KUKA KRL program: MyProgram_143().src

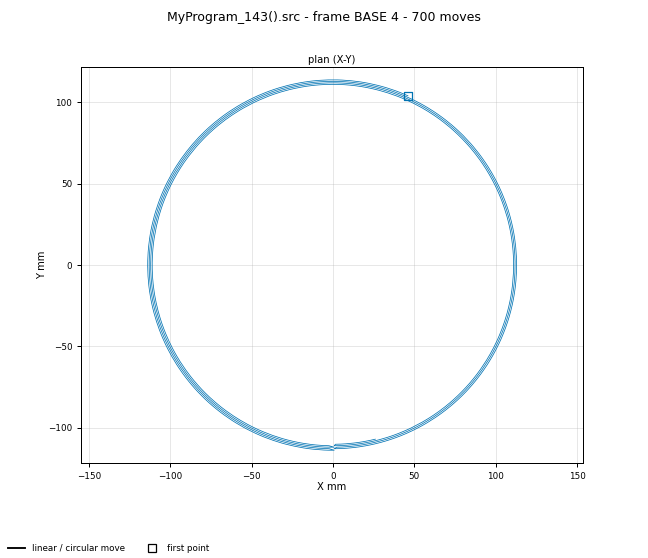
[picture p0: tool path of MyProgram_143().src in frame BASE 4, 700 of 700 moves have a stored position in this frame; points joined in program order, loops and branches not executed]
&ACCESS RVP
&REL 1
&PARAM TEMPLATE = C:\KRC\Roboter\Template\vorgabe
&PARAM EDITMASK = *
DEF MyProgram_143()
; ---- Setting reference (Base) ----
$BASE = BASE_DATA[4]

; --------------------------
; ---- Setting tool (TCP) ----
$TOOL = TOOL_DATA[3]
; --------------------------

$VEL.CP = VEL_APROX_PRINT
Startdeposition()
$VEL.CP = VEL_PRINT
LIN {X 46.1165,Y 104.0371,Z 114,A 62.0939,B 24.9325,C -1.8981,E1 25.0637,E2 383.7056} C_DIS
LIN {X 43.2178,Y 105.2725,Z 114,A 63.5467,B 24.9328,C -1.8939,E1 25.06,E2 382.2661} C_DIS
LIN {X 40.9561,Y 106.1746,Z 114,A 64.7702,B 24.9327,C -1.895,E1 25.0568,E2 381.0428} C_DIS
LIN {X 38.0003,Y 107.2663,Z 114,A 66.3534,B 24.9326,C -1.8963,E1 25.0527,E2 379.4597} C_DIS
LIN {X 35.3564,Y 108.1666,Z 114,A 67.7569,B 24.9326,C -1.8974,E1 25.0489,E2 378.0564} C_DIS
LIN {X 33.0344,Y 108.8999,Z 114,A 69.1112,B 24.932,C -1.9039,E1 25.0453,E2 376.689} C_DIS
LIN {X 30.3519,Y 109.6778,Z 114,A 70.5154,B 24.932,C -1.9048,E1 25.0415,E2 375.2851} C_DIS
LIN {X 27.6512,Y 110.3896,Z 114,A 71.9198,B 24.932,C -1.9055,E1 25.0377,E2 373.881} C_DIS
LIN {X 24.584,Y 111.1112,Z 114,A 73.211,B 24.9328,C -1.8936,E1 25.0343,E2 372.6199} C_DIS
LIN {X 22.2013,Y 111.6134,Z 114,A 74.5993,B 24.9322,C -1.9011,E1 25.0304,E2 371.2154} C_DIS
LIN {X 19.4555,Y 112.1246,Z 114,A 76.0045,B 24.9322,C -1.9016,E1 25.0266,E2 369.8105} C_DIS
LIN {X 16.6979,Y 112.5683,Z 114,A 77.5399,B 24.9318,C -1.9077,E1 25.0223,E2 368.2623} C_DIS
LIN {X 13.5748,Y 112.9859,Z 114,A 78.8318,B 24.9327,C -1.8953,E1 25.0188,E2 367.0007} C_DIS
LIN {X 11.1544,Y 113.2521,Z 114,A 80.3513,B 24.9317,C -1.9081,E1 25.0145,E2 365.4519} C_DIS
LIN {X 8.0145,Y 113.5158,Z 114,A 81.8072,B 24.9321,C -1.9026,E1 25.0105,E2 364.0098} C_DIS
LIN {X 5.5839,Y 113.663,Z 114,A 83.1636,B 24.9317,C -1.9081,E1 25.0067,E2 362.6407} C_DIS
LIN {X 2.7928,Y 113.7658,Z 114,A 84.4401,B 24.9322,C -1.9024,E1 25.0032,E2 361.3781} C_DIS
LIN {X -0.358,Y 113.7978,Z 114,A 86.0421,B 24.9322,C -1.9028,E1 24.9987,E2 359.7753} C_DIS
LIN {X -2.7928,Y 113.7658,Z 114,A 87.3841,B 24.9318,C -1.9074,E1 24.9949,E2 358.4222} C_DIS
LIN {X -5.7875,Y 113.6517,Z 114,A 88.6706,B 24.9325,C -1.8975,E1 24.9914,E2 357.159} C_DIS
LIN {X -8.3717,Y 113.4917,Z 114,A 90.1989,B 24.9319,C -1.9064,E1 24.9871,E2 355.6088} C_DIS
LIN {X -11.5104,Y 113.2148,Z 114,A 91.4931,B 24.9328,C -1.8933,E1 24.9835,E2 354.3452} C_DIS
LIN {X -14.2853,Y 112.8982,Z 114,A 93.065,B 24.9324,C -1.8995,E1 24.9791,E2 352.7575} C_DIS
LIN {X -17.0517,Y 112.5136,Z 114,A 94.473,B 24.9324,C -1.8986,E1 24.9753,E2 351.3504} C_DIS
LIN {X -19.8078,Y 112.0613,Z 114,A 95.8815,B 24.9324,C -1.8977,E1 24.9714,E2 349.9428} C_DIS
LIN {X -22.5519,Y 111.5414,Z 114,A 97.3152,B 24.9324,C -1.8977,E1 24.9674,E2 348.5075} C_DIS
LIN {X -24.9337,Y 111.0349,Z 114,A 98.5186,B 24.9326,C -1.8956,E1 24.9642,E2 347.3074} C_DIS
LIN {X -28.04,Y 110.2897,Z 114,A 100.1157,B 24.9328,C -1.8936,E1 24.9598,E2 345.7129} C_DIS
LIN {X -30.7893,Y 109.5538,Z 114,A 101.5344,B 24.9329,C -1.8915,E1 24.956,E2 344.2969} C_DIS
LIN {X -33.3763,Y 108.7938,Z 114,A 102.9287,B 24.9329,C -1.8915,E1 24.9523,E2 342.9003} C_DIS
LIN {X -36.0362,Y 107.942,Z 114,A 104.1731,B 24.9335,C -1.8831,E1 24.949,E2 341.6736} C_DIS
LIN {X -38.6744,Y 107.0251,Z 114,A 105.7474,B 24.9332,C -1.8883,E1 24.9449,E2 340.0839} C_DIS
LIN {X -41.2893,Y 106.0437,Z 114,A 107.1576,B 24.9332,C -1.8866,E1 24.9412,E2 338.6748} C_DIS
LIN {X -43.8793,Y 104.9985,Z 114,A 108.5683,B 24.9334,C -1.8848,E1 24.9375,E2 337.2652} C_DIS
LIN {X -46.1165,Y 104.0371,Z 114,A 109.7983,B 24.9335,C -1.8831,E1 24.9344,E2 336.0362} C_DIS
LIN {X -48.6835,Y 102.8607,Z 114,A 111.3437,B 24.9333,C -1.886,E1 24.9305,E2 334.4801} C_DIS
LIN {X -51.4845,Y 101.4861,Z 114,A 112.8012,B 24.9338,C -1.8788,E1 24.9269,E2 333.0359} C_DIS
LIN {X -53.9596,Y 100.192,Z 114,A 114.2127,B 24.934,C -1.8767,E1 24.9234,E2 331.6255} C_DIS
LIN {X -56.0918,Y 99.0159,Z 114,A 115.4434,B 24.9341,C -1.8747,E1 24.9204,E2 330.3961} C_DIS
LIN {X -58.8108,Y 97.4236,Z 114,A 117.036,B 24.9343,C -1.8721,E1 24.9166,E2 328.8048} C_DIS
LIN {X -61.184,Y 95.951,Z 114,A 118.2834,B 24.9349,C -1.8629,E1 24.9137,E2 327.5752} C_DIS
LIN {X -63.2239,Y 94.6213,Z 114,A 119.8102,B 24.9343,C -1.8728,E1 24.91,E2 326.0199} C_DIS
LIN {X -65.8184,Y 92.8333,Z 114,A 121.2145,B 24.935,C -1.8622,E1 24.9069,E2 324.636} C_DIS
LIN {X -68.0768,Y 91.1901,Z 114,A 122.5208,B 24.9355,C -1.8552,E1 24.904,E2 323.3418} C_DIS
LIN {X -70.2942,Y 89.4919,Z 114,A 124.098,B 24.9352,C -1.8591,E1 24.9004,E2 321.7495} C_DIS
LIN {X -72.194,Y 87.9686,Z 114,A 125.3301,B 24.9354,C -1.8566,E1 24.8978,E2 320.5187} C_DIS
LIN {X -74.3311,Y 86.1704,Z 114,A 126.874,B 24.9352,C -1.859,E1 24.8945,E2 318.963} C_DIS
LIN {X -76.4234,Y 84.3203,Z 114,A 128.1561,B 24.9358,C -1.8507,E1 24.8918,E2 317.6955} C_DIS
LIN {X -78.4697,Y 82.4194,Z 114,A 129.7007,B 24.9356,C -1.853,E1 24.8887,E2 316.1392} C_DIS
LIN {X -80.7204,Y 80.2141,Z 114,A 131.1644,B 24.9362,C -1.8442,E1 24.8858,E2 314.6902} C_DIS
LIN {X -82.4194,Y 78.4697,Z 114,A 132.564,B 24.936,C -1.8482,E1 24.8831,E2 313.2751} C_DIS
LIN {X -84.559,Y 76.1567,Z 114,A 133.9922,B 24.9367,C -1.8378,E1 24.8804,E2 311.8653} C_DIS
LIN {X -86.1704,Y 74.3311,Z 114,A 135.2253,B 24.9369,C -1.8349,E1 24.8782,E2 310.6336} C_DIS
LIN {X -88.194,Y 71.9159,Z 114,A 136.6561,B 24.9376,C -1.8245,E1 24.8756,E2 309.2209} C_DIS
LIN {X -89.7139,Y 70.0134,Z 114,A 138.0538,B 24.9374,C -1.8281,E1 24.8732,E2 307.8081} C_DIS
LIN {X -91.6165,Y 67.5018,Z 114,A 139.4849,B 24.9381,C -1.8176,E1 24.8708,E2 306.3952} C_DIS
LIN {X -93.0412,Y 65.527,Z 114,A 141.0139,B 24.9375,C -1.8263,E1 24.8683,E2 304.8379} C_DIS
LIN {X -94.8183,Y 62.9251,Z 114,A 142.4789,B 24.9381,C -1.817,E1 24.866,E2 303.3877} C_DIS
LIN {X -96.1444,Y 60.8828,Z 114,A 143.8436,B 24.938,C -1.8191,E1 24.864,E2 302.0113} C_DIS
LIN {X -97.6096,Y 58.5049,Z 114,A 145.1278,B 24.9386,C -1.8101,E1 24.8621,E2 300.7418} C_DIS
LIN {X -99.1905,Y 55.7793,Z 114,A 146.5592,B 24.9393,C -1.7993,E1 24.8602,E2 299.3286} C_DIS
LIN {X -100.5295,Y 53.3282,Z 114,A 147.9748,B 24.9396,C -1.7956,E1 24.8583,E2 297.9145} C_DIS
LIN {X -101.649,Y 51.1658,Z 114,A 149.3733,B 24.9394,C -1.7988,E1 24.8565,E2 296.501} C_DIS
LIN {X -102.874,Y 48.6558,Z 114,A 150.7887,B 24.9396,C -1.7949,E1 24.8548,E2 295.0871} C_DIS
LIN {X -104.0371,Y 46.1165,Z 114,A 152.3355,B 24.9396,C -1.7962,E1 24.853,E2 293.5286} C_DIS
LIN {X -105.1375,Y 43.5494,Z 114,A 153.6201,B 24.9401,C -1.787,E1 24.8516,E2 292.2588} C_DIS
LIN {X -106.1746,Y 40.9561,Z 114,A 155.0356,B 24.9404,C -1.7831,E1 24.8502,E2 290.8448} C_DIS
LIN {X -107.2085,Y 38.1651,Z 114,A 156.6062,B 24.9405,C -1.7813,E1 24.8487,E2 289.2696} C_DIS
LIN {X -108.1666,Y 35.3564,Z 114,A 157.8837,B 24.9414,C -1.768,E1 24.8476,E2 288.0165} C_DIS
LIN {X -108.8999,Y 33.0344,Z 114,A 159.2832,B 24.9412,C -1.771,E1 24.8464,E2 286.6019} C_DIS
LIN {X -109.7859,Y 29.9514,Z 114,A 160.7183,B 24.942,C -1.7587,E1 24.8453,E2 285.1876} C_DIS
LIN {X -110.4745,Y 27.3034,Z 114,A 162.1316,B 24.9422,C -1.7557,E1 24.8444,E2 283.7732} C_DIS
LIN {X -111.1112,Y 24.584,Z 114,A 163.7041,B 24.9421,C -1.7578,E1 24.8434,E2 282.1865} C_DIS
LIN {X -111.6811,Y 21.8498,Z 114,A 165.1331,B 24.9423,C -1.7542,E1 24.8426,E2 280.7577} C_DIS
LIN {X -112.1837,Y 19.1024,Z 114,A 166.3797,B 24.943,C -1.7433,E1 24.842,E2 279.5296} C_DIS
LIN {X -112.6187,Y 16.3435,Z 114,A 167.7956,B 24.9433,C -1.7391,E1 24.8414,E2 278.1152} C_DIS
LIN {X -112.9859,Y 13.5748,Z 114,A 169.2121,B 24.9436,C -1.735,E1 24.8409,E2 276.7003} C_DIS
LIN {X -113.2521,Y 11.1544,Z 114,A 170.6117,B 24.9434,C -1.7379,E1 24.8405,E2 275.2854} C_DIS
LIN {X -113.5158,Y 8.0145,Z 114,A 172.209,B 24.9437,C -1.7332,E1 24.8401,E2 273.6896} C_DIS
LIN {X -113.6762,Y 5.2757,Z 114,A 173.6173,B 24.9439,C -1.7297,E1 24.8399,E2 272.2811} C_DIS
LIN {X -113.7658,Y 2.7928,Z 114,A 175.0421,B 24.9437,C -1.7326,E1 24.8399,E2 270.8409} C_DIS
LIN {X -113.7945,Y -0.969,Z 114,A 176.8249,B 24.9444,C -1.722,E1 24.8399,E2 269.0726} C_DIS
LIN {X -113.7006,Y -4.7094,Z 114,A 178.4247,B 24.9455,C -1.7046,E1 24.8399,E2 267.5046} C_DIS
LIN {X -113.5859,Y -6.9783,Z 114,A 179.9475,B 24.9448,C -1.716,E1 24.8402,E2 265.9456} C_DIS
LIN {X -113.3475,Y -10.1202,Z 114,A -178.5862,B 24.9455,C -1.7061,E1 24.8405,E2 264.494} C_DIS
LIN {X -113.1067,Y -12.5433,Z 114,A -177.2205,B 24.9453,C -1.7077,E1 24.8409,E2 263.1162} C_DIS
LIN {X -112.7144,Y -15.6697,Z 114,A -175.7543,B 24.946,C -1.6979,E1 24.8415,E2 261.6647} C_DIS
LIN {X -112.2959,Y -18.4311,Z 114,A -174.503,B 24.9466,C -1.6873,E1 24.842,E2 260.4313} C_DIS
LIN {X -111.8774,Y -20.8299,Z 114,A -172.9727,B 24.9461,C -1.6955,E1 24.8428,E2 258.8723} C_DIS
LIN {X -111.3326,Y -23.5693,Z 114,A -171.5211,B 24.9463,C -1.6929,E1 24.8436,E2 257.4183} C_DIS
LIN {X -110.7206,Y -26.2944,Z 114,A -170.1412,B 24.9466,C -1.6875,E1 24.8445,E2 256.0432} C_DIS
LIN {X -109.9486,Y -29.3493,Z 114,A -168.6752,B 24.9472,C -1.6778,E1 24.8455,E2 254.5919} C_DIS
LIN {X -109.1952,Y -32.0387,Z 114,A -167.4243,B 24.9479,C -1.6673,E1 24.8464,E2 253.3588} C_DIS
LIN {X -108.3987,Y -34.639,Z 114,A -166.0121,B 24.9481,C -1.6648,E1 24.8476,E2 251.9442} C_DIS
LIN {X -107.6102,Y -37.0203,Z 114,A -164.61,B 24.948,C -1.6666,E1 24.8489,E2 250.53} C_DIS
LIN {X -106.6692,Y -39.6501,Z 114,A -163.0638,B 24.9479,C -1.668,E1 24.8504,E2 248.9716} C_DIS
LIN {X -105.5291,Y -42.5875,Z 114,A -161.5985,B 24.9485,C -1.6585,E1 24.8519,E2 247.5207} C_DIS
LIN {X -104.4521,Y -45.1645,Z 114,A -160.1215,B 24.9485,C -1.6573,E1 24.8535,E2 246.0385} C_DIS
LIN {X -102.874,Y -48.6558,Z 114,A -158.1112,B 24.9487,C -1.655,E1 24.8559,E2 244.0226} C_DIS
LIN {X -101.4861,Y -51.4845,Z 114,A -156.6461,B 24.9492,C -1.6457,E1 24.8577,E2 242.5718} C_DIS
LIN {X -100.192,Y -53.9596,Z 114,A -155.2312,B 24.9495,C -1.6422,E1 24.8595,E2 241.1579} C_DIS
LIN {X -99.0159,Y -56.0918,Z 114,A -153.998,B 24.9497,C -1.6391,E1 24.8612,E2 239.9256} C_DIS
LIN {X -97.3228,Y -58.9767,Z 114,A -152.3668,B 24.9501,C -1.6325,E1 24.8635,E2 238.3017} C_DIS
LIN {X -95.951,Y -61.184,Z 114,A -151.1167,B 24.9504,C -1.6267,E1 24.8654,E2 237.0591} C_DIS
LIN {X -94.6213,Y -63.2239,Z 114,A -149.6243,B 24.95,C -1.6343,E1 24.8677,E2 235.541} C_DIS
LIN {X -92.2301,Y -66.6638,Z 114,A -147.5035,B 24.9502,C -1.6295,E1 24.8711,E2 233.4214} C_DIS
LIN {X -90.5663,Y -68.9072,Z 114,A -146.09,B 24.9504,C -1.6263,E1 24.8735,E2 232.0086} C_DIS
LIN {X -88.8479,Y -71.109,Z 114,A -144.8071,B 24.951,C -1.6179,E1 24.8757,E2 230.7398} C_DIS
LIN {X -86.8439,Y -73.5405,Z 114,A -143.377,B 24.9516,C -1.6078,E1 24.8782,E2 229.3271} C_DIS
LIN {X -85.013,Y -75.6497,Z 114,A -141.7994,B 24.9513,C -1.6116,E1 24.8812,E2 227.7334} C_DIS
LIN {X -83.1309,Y -77.7132,Z 114,A -140.3002,B 24.9513,C -1.6122,E1 24.884,E2 226.2259} C_DIS
LIN {X -80.4688,Y -80.4688,Z 114,A -138.4479,B 24.9517,C -1.6049,E1 24.8876,E2 224.3833} C_DIS
LIN {X -78.4697,Y -82.4194,Z 114,A -137.0355,B 24.9519,C -1.6022,E1 24.8905,E2 222.9714} C_DIS
LIN {X -76.4234,Y -84.3203,Z 114,A -135.4925,B 24.9517,C -1.605,E1 24.8937,E2 221.4155} C_DIS
LIN {X -74.3311,Y -86.1704,Z 114,A -134.0244,B 24.9517,C -1.6048,E1 24.8968,E2 219.9421} C_DIS
LIN {X -71.109,Y -88.8479,Z 114,A -131.9623,B 24.9521,C -1.5989,E1 24.9012,E2 217.8863} C_DIS
LIN {X -68.9072,Y -90.5663,Z 114,A -130.5508,B 24.9522,C -1.5966,E1 24.9044,E2 216.4751} C_DIS
LIN {X -66.6638,Y -92.2301,Z 114,A -129.2697,B 24.9527,C -1.5889,E1 24.9072,E2 215.2078} C_DIS
LIN {X -64.0839,Y -94.039,Z 114,A -127.6777,B 24.9528,C -1.5865,E1 24.9109,E2 213.6161} C_DIS
LIN {X -62.058,Y -95.39,Z 114,A -126.4471,B 24.9529,C -1.5848,E1 24.9137,E2 212.3856} C_DIS
LIN {X -59.6983,Y -96.8843,Z 114,A -124.906,B 24.9527,C -1.5883,E1 24.9174,E2 210.8313} C_DIS
LIN {X -56.9923,Y -98.4985,Z 114,A -123.6091,B 24.9536,C -1.5739,E1 24.9205,E2 209.5648} C_DIS
LIN {X -54.8725,Y -99.6968,Z 114,A -122.2152,B 24.9533,C -1.5792,E1 24.9239,E2 208.1543} C_DIS
LIN {X -52.4093,Y -101.0134,Z 114,A -120.8052,B 24.9533,C -1.5775,E1 24.9274,E2 206.7443} C_DIS
LIN {X -49.5919,Y -102.4242,Z 114,A -119.3037,B 24.9537,C -1.572,E1 24.9311,E2 205.2519} C_DIS
LIN {X -47.3897,Y -103.4634,Z 114,A -117.9855,B 24.9536,C -1.5744,E1 24.9345,E2 203.9246} C_DIS
LIN {X -44.8363,Y -104.5952,Z 114,A -116.5759,B 24.9536,C -1.573,E1 24.9381,E2 202.515} C_DIS
LIN {X -42.2559,Y -105.664,Z 114,A -115.0363,B 24.9534,C -1.5773,E1 24.9421,E2 200.9619} C_DIS
LIN {X -39.0676,Y -106.8817,Z 114,A -113.4085,B 24.9537,C -1.5719,E1 24.9464,E2 199.3436} C_DIS
LIN {X -36.6811,Y -107.7245,Z 114,A -112.1681,B 24.9539,C -1.5694,E1 24.9496,E2 198.1068} C_DIS
LIN {X -34.0264,Y -108.5923,Z 114,A -110.9232,B 24.9543,C -1.5614,E1 24.9529,E2 196.8785} C_DIS
LIN {X -31.6956,Y -109.297,Z 114,A -109.4288,B 24.9537,C -1.572,E1 24.957,E2 195.3565} C_DIS
LIN {X -29.0037,Y -110.042,Z 114,A -107.9933,B 24.9537,C -1.5724,E1 24.9609,E2 193.9179} C_DIS
LIN {X -25.9456,Y -110.8012,Z 114,A -106.5353,B 24.9541,C -1.566,E1 24.9648,E2 192.473} C_DIS
LIN {X -23.5693,Y -111.3326,Z 114,A -105.1778,B 24.9538,C -1.5711,E1 24.9685,E2 191.1018} C_DIS
LIN {X -20.4423,Y -111.9472,Z 114,A -103.8822,B 24.9546,C -1.5572,E1 24.972,E2 189.8378} C_DIS
LIN {X -18.0781,Y -112.3549,Z 114,A -102.4935,B 24.9541,C -1.5646,E1 24.9759,E2 188.4303} C_DIS
LIN {X -15.3153,Y -112.7648,Z 114,A -100.9564,B 24.9538,C -1.57,E1 24.9801,E2 186.8792} C_DIS
LIN {X -11.9787,Y -113.1658,Z 114,A -99.452,B 24.9543,C -1.5616,E1 24.9843,E2 185.3937} C_DIS
LIN {X -8.0145,Y -113.5158,Z 114,A -97.3901,B 24.9542,C -1.5641,E1 24.99,E2 183.325} C_DIS
LIN {X -5.5839,Y -113.663,Z 114,A -96.0341,B 24.9538,C -1.5698,E1 24.9939,E2 181.955} C_DIS
LIN {X -2.7928,Y -113.7658,Z 114,A -94.7582,B 24.9542,C -1.5643,E1 24.9974,E2 180.692} C_DIS
LIN {X 0.7991,Y -113.7938,Z 114,A -93.1524,B 24.9546,C -1.5559,E1 25.0018,E2 179.1062} C_DIS
Enddeposition()
LIN {X 0.7991,Y -113.7938,Z 114,A -93.1524,B 24.9546,C -1.5559,E1 25.0018,E2 179.1062} C_DIS
Startdeposition()
$VEL.CP = VEL_PRINT
LIN {X -2.2586,Y -112.8565,Z 114,A -95.1963,B 24.955,C -1.5503,E1 24.9961,E2 181.1633} C_DIS
LIN {X -9.0135,Y -112.5185,Z 114,A -98.6101,B 24.955,C -1.551,E1 24.9866,E2 184.5765} C_DIS
LIN {X -13.6469,Y -112.0522,Z 114,A -100.9708,B 24.955,C -1.5513,E1 24.98,E2 186.9379} C_DIS
LIN {X -18.5418,Y -111.3457,Z 114,A -103.5657,B 24.955,C -1.5484,E1 24.9728,E2 189.5418} C_DIS
LIN {X -22.4378,Y -110.6268,Z 114,A -105.6155,B 24.9551,C -1.5475,E1 24.9672,E2 191.596} C_DIS
LIN {X -26.0122,Y -109.8427,Z 114,A -107.4525,B 24.9551,C -1.5493,E1 24.9622,E2 193.4312} C_DIS
LIN {X -29.3354,Y -109.0005,Z 114,A -109.1292,B 24.9548,C -1.553,E1 24.9577,E2 195.1015} C_DIS
LIN {X -31.7632,Y -108.3185,Z 114,A -110.5257,B 24.955,C -1.549,E1 24.9539,E2 196.5098} C_DIS
LIN {X -35.5601,Y -107.1328,Z 114,A -112.4447,B 24.9547,C -1.5547,E1 24.9488,E2 198.4187} C_DIS
LIN {X -38.7299,Y -106.0267,Z 114,A -114.1848,B 24.9547,C -1.5547,E1 24.9442,E2 200.1622} C_DIS
LIN {X -42.313,Y -104.6487,Z 114,A -116.1255,B 24.9546,C -1.557,E1 24.9392,E2 202.1019} C_DIS
LIN {X -46.2152,Y -102.9847,Z 114,A -118.2734,B 24.9544,C -1.5595,E1 24.9337,E2 204.2487} C_DIS
LIN {X -48.99,Y -101.694,Z 114,A -119.7945,B 24.9542,C -1.5627,E1 24.9298,E2 205.7662} C_DIS
LIN {X -52.1714,Y -100.1002,Z 114,A -121.6226,B 24.9542,C -1.5641,E1 24.9253,E2 207.5959} C_DIS
LIN {X -54.6205,Y -98.7851,Z 114,A -123.1671,B 24.9544,C -1.5605,E1 24.9215,E2 209.1532} C_DIS
LIN {X -58.226,Y -96.7038,Z 114,A -125.2381,B 24.9541,C -1.5653,E1 24.9165,E2 211.2192} C_DIS
LIN {X -61.5631,Y -94.6156,Z 114,A -127.1227,B 24.9536,C -1.573,E1 24.9121,E2 213.0914} C_DIS
LIN {X -63.5831,Y -93.2683,Z 114,A -128.4203,B 24.9536,C -1.5724,E1 24.9091,E2 214.3948} C_DIS
LIN {X -66.6222,Y -91.1216,Z 114,A -130.2576,B 24.9534,C -1.5777,E1 24.9049,E2 216.2259} C_DIS
LIN {X -69.0307,Y -89.311,Z 114,A -131.7931,B 24.9532,C -1.5802,E1 24.9015,E2 217.761} C_DIS
LIN {X -71.4837,Y -87.3615,Z 114,A -133.5417,B 24.9534,C -1.5767,E1 24.8977,E2 219.5244} C_DIS
LIN {X -74.0275,Y -85.2155,Z 114,A -135.1616,B 24.9531,C -1.5828,E1 24.8943,E2 221.1361} C_DIS
LIN {X -76.6052,Y -82.9063,Z 114,A -136.8906,B 24.9528,C -1.5875,E1 24.8907,E2 222.861} C_DIS
LIN {X -79.2467,Y -80.3843,Z 114,A -138.7926,B 24.9527,C -1.5894,E1 24.8869,E2 224.7663} C_DIS
LIN {X -81.9311,Y -77.6476,Z 114,A -140.7693,B 24.9525,C -1.5924,E1 24.883,E2 226.7444} C_DIS
LIN {X -84.589,Y -74.7448,Z 114,A -142.8598,B 24.9525,C -1.5932,E1 24.8791,E2 228.8423} C_DIS
LIN {X -87.2958,Y -71.5648,Z 114,A -145.0018,B 24.9522,C -1.5973,E1 24.8753,E2 230.9844} C_DIS
LIN {X -89.4995,Y -68.786,Z 114,A -146.6681,B 24.9516,C -1.607,E1 24.8724,E2 232.6355} C_DIS
LIN {X -91.6911,Y -65.8371,Z 114,A -148.3274,B 24.9508,C -1.6198,E1 24.8697,E2 234.2722} C_DIS
LIN {X -93.0166,Y -63.9524,Z 114,A -149.7858,B 24.9514,C -1.6113,E1 24.8674,E2 235.7581} C_DIS
LIN {X -94.5965,Y -61.5921,Z 114,A -151.1105,B 24.9508,C -1.6196,E1 24.8654,E2 237.0696} C_DIS
LIN {X -96.2719,Y -58.9366,Z 114,A -152.8227,B 24.9508,C -1.6192,E1 24.8628,E2 238.7916} C_DIS
LIN {X -98.1671,Y -55.7247,Z 114,A -154.6317,B 24.9504,C -1.6276,E1 24.8603,E2 240.59} C_DIS
LIN {X -100.8755,Y -50.6571,Z 114,A -157.6127,B 24.95,C -1.6331,E1 24.8564,E2 243.5737} C_DIS
LIN {X -102.3686,Y -47.564,Z 114,A -159.3935,B 24.9498,C -1.6366,E1 24.8543,E2 245.3558} C_DIS
LIN {X -103.7319,Y -44.5169,Z 114,A -161.1653,B 24.9497,C -1.6384,E1 24.8523,E2 247.1331} C_DIS
LIN {X -104.9067,Y -41.6706,Z 114,A -162.6469,B 24.9492,C -1.6462,E1 24.8507,E2 248.6044} C_DIS
LIN {X -105.9693,Y -38.8872,Z 114,A -164.1989,B 24.949,C -1.6491,E1 24.8492,E2 250.1582} C_DIS
LIN {X -107.043,Y -35.8264,Z 114,A -165.8973,B 24.9489,C -1.652,E1 24.8477,E2 251.8594} C_DIS
LIN {X -108.0614,Y -32.6277,Z 114,A -168.1598,B 24.9499,C -1.6355,E1 24.8458,E2 254.1742} C_DIS
LIN {X -109.2232,Y -28.4979,Z 114,A -169.7983,B 24.9482,C -1.6631,E1 24.8447,E2 255.7565} C_DIS
LIN {X -110.1558,Y -24.6524,Z 114,A -171.7438,B 24.9476,C -1.6718,E1 24.8434,E2 257.6927} C_DIS
LIN {X -110.7486,Y -21.8326,Z 114,A -173.0922,B 24.9471,C -1.6808,E1 24.8427,E2 259.0275} C_DIS
LIN {X -111.2957,Y -18.841,Z 114,A -174.626,B 24.9467,C -1.6861,E1 24.8419,E2 260.5579} C_DIS
LIN {X -111.7711,Y -15.7763,Z 114,A -176.4489,B 24.947,C -1.6814,E1 24.8412,E2 262.4027} C_DIS
LIN {X -112.2153,Y -12.2317,Z 114,A -178.0389,B 24.9461,C -1.6959,E1 24.8407,E2 263.9678} C_DIS
LIN {X -112.5139,Y -9.0719,Z 114,A -179.8355,B 24.9462,C -1.6939,E1 24.8402,E2 265.78} C_DIS
LIN {X -112.7457,Y -5.5256,Z 114,A 178.2019,B 24.9462,C -1.6935,E1 24.8399,E2 267.7553} C_DIS
LIN {X -112.8722,Y -1.397,Z 114,A 176.1161,B 24.9458,C -1.7007,E1 24.8398,E2 269.8364} C_DIS
LIN {X -112.8551,Y 2.3368,Z 114,A 174.3952,B 24.945,C -1.7136,E1 24.8398,E2 271.5369} C_DIS
LIN {X -112.7327,Y 5.7632,Z 114,A 172.7548,B 24.9444,C -1.7231,E1 24.84,E2 273.1644} C_DIS
LIN {X -112.5317,Y 8.8494,Z 114,A 170.9857,B 24.9445,C -1.7205,E1 24.8404,E2 274.9504} C_DIS
LIN {X -112.1713,Y 12.6301,Z 114,A 169.0198,B 24.9442,C -1.7253,E1 24.8409,E2 276.9168} C_DIS
LIN {X -111.6851,Y 16.382,Z 114,A 167.0194,B 24.944,C -1.7284,E1 24.8417,E2 278.9217} C_DIS
LIN {X -111.1787,Y 19.5236,Z 114,A 165.3457,B 24.9438,C -1.7314,E1 24.8425,E2 280.5982} C_DIS
LIN {X -110.3652,Y 23.6924,Z 114,A 163.2697,B 24.9432,C -1.7414,E1 24.8437,E2 282.6625} C_DIS
LIN {X -109.5151,Y 27.3588,Z 114,A 161.1089,B 24.9434,C -1.7379,E1 24.8451,E2 284.8445} C_DIS
LIN {X -108.2752,Y 31.9089,Z 114,A 159.1024,B 24.9419,C -1.7605,E1 24.8466,E2 286.8087} C_DIS
LIN {X -107.2912,Y 35.0758,Z 114,A 157.205,B 24.9421,C -1.7575,E1 24.8482,E2 288.7242} C_DIS
LIN {X -106.422,Y 37.6311,Z 114,A 155.3289,B 24.9431,C -1.7422,E1 24.85,E2 290.6472} C_DIS
LIN {X -104.9357,Y 41.5967,Z 114,A 153.3141,B 24.9423,C -1.7541,E1 24.8521,E2 292.6452} C_DIS
LIN {X -103.5701,Y 44.8882,Z 114,A 151.811,B 24.9412,C -1.7714,E1 24.8537,E2 294.1152} C_DIS
LIN {X -101.9941,Y 48.3653,Z 114,A 150.106,B 24.9402,C -1.7863,E1 24.8556,E2 295.7941} C_DIS
LIN {X -100.589,Y 51.2206,Z 114,A 148.4035,B 24.9401,C -1.7877,E1 24.8578,E2 297.5022} C_DIS
LIN {X -99.0805,Y 54.0815,Z 114,A 146.6333,B 24.9401,C -1.7876,E1 24.8601,E2 299.2822} C_DIS
LIN {X -97.4137,Y 57.0303,Z 114,A 144.5089,B 24.9408,C -1.7769,E1 24.8632,E2 301.4431} C_DIS
LIN {X -95.5003,Y 60.1794,Z 114,A 143.0585,B 24.9394,C -1.7985,E1 24.8652,E2 302.8494} C_DIS
LIN {X -93.6718,Y 62.9873,Z 114,A 141.3181,B 24.9392,C -1.8017,E1 24.8679,E2 304.5908} C_DIS
LIN {X -91.4817,Y 66.1305,Z 114,A 139.328,B 24.9389,C -1.8053,E1 24.8711,E2 306.5821} C_DIS
LIN {X -89.4267,Y 68.8806,Z 114,A 137.7955,B 24.938,C -1.8183,E1 24.8737,E2 308.091} C_DIS
LIN {X -87.085,Y 71.8196,Z 114,A 135.6803,B 24.9382,C -1.8152,E1 24.8774,E2 310.2235} C_DIS
LIN {X -84.6596,Y 74.664,Z 114,A 133.7205,B 24.9381,C -1.8176,E1 24.881,E2 312.1863} C_DIS
LIN {X -81.997,Y 77.5775,Z 114,A 131.7125,B 24.9377,C -1.8225,E1 24.8848,E2 314.1915} C_DIS
LIN {X -79.2984,Y 80.3332,Z 114,A 129.8833,B 24.9371,C -1.8323,E1 24.8884,E2 316.0051} C_DIS
LIN {X -76.5557,Y 82.9518,Z 114,A 127.8785,B 24.937,C -1.8337,E1 24.8925,E2 318.0148} C_DIS
LIN {X -73.5611,Y 85.6192,Z 114,A 125.8041,B 24.9368,C -1.8368,E1 24.8968,E2 320.09} C_DIS
LIN {X -71.2356,Y 87.5626,Z 114,A 124.4734,B 24.936,C -1.8485,E1 24.8997,E2 321.398} C_DIS
LIN {X -68.5761,Y 89.6613,Z 114,A 122.5677,B 24.9362,C -1.8447,E1 24.9039,E2 323.3196} C_DIS
LIN {X -65.7243,Y 91.7716,Z 114,A 120.9294,B 24.9355,C -1.8549,E1 24.9076,E2 324.9394} C_DIS
LIN {X -63.3156,Y 93.4495,Z 114,A 119.4932,B 24.9351,C -1.8601,E1 24.9108,E2 326.3682} C_DIS
LIN {X -61.3117,Y 94.7771,Z 114,A 118.2307,B 24.9351,C -1.8607,E1 24.9138,E2 327.6332} C_DIS
LIN {X -58.7388,Y 96.3921,Z 114,A 116.5385,B 24.9353,C -1.8576,E1 24.9178,E2 329.3381} C_DIS
LIN {X -56.6184,Y 97.6535,Z 114,A 114.6159,B 24.937,C -1.8332,E1 24.9227,E2 331.3246} C_DIS
LIN {X -52.6966,Y 99.8236,Z 114,A 112.4916,B 24.9363,C -1.843,E1 24.9278,E2 333.4314} C_DIS
LIN {X -49.2421,Y 101.5728,Z 114,A 111.1622,B 24.9343,C -1.8717,E1 24.931,E2 334.6962} C_DIS
LIN {X -46.4263,Y 102.8896,Z 114,A 109.3838,B 24.9347,C -1.866,E1 24.9356,E2 336.4924} C_DIS
LIN {X -41.5441,Y 104.9564,Z 114,A 106.7183,B 24.9344,C -1.8708,E1 24.9424,E2 339.1525} C_DIS
LIN {X -38.1852,Y 106.2254,Z 114,A 104.9718,B 24.934,C -1.8763,E1 24.947,E2 340.8895} C_DIS
LIN {X -35.1193,Y 107.2775,Z 114,A 103.468,B 24.9335,C -1.8841,E1 24.9509,E2 342.3777} C_DIS
LIN {X -31.7358,Y 108.3266,Z 114,A 101.3455,B 24.9342,C -1.8729,E1 24.9567,E2 344.5304} C_DIS
LIN {X -27.4808,Y 109.4846,Z 114,A 99.1741,B 24.9339,C -1.8779,E1 24.9625,E2 346.6932} C_DIS
LIN {X -24.2336,Y 110.2471,Z 114,A 97.5558,B 24.9336,C -1.8825,E1 24.9669,E2 348.3026} C_DIS
LIN {X -21.6518,Y 110.7834,Z 114,A 96.1851,B 24.9336,C -1.8823,E1 24.9706,E2 349.6754} C_DIS
LIN {X -18.5129,Y 111.3506,Z 114,A 94.4953,B 24.9337,C -1.8806,E1 24.9753,E2 351.3709} C_DIS
LIN {X -15.1856,Y 111.855,Z 114,A 92.7805,B 24.9337,C -1.8814,E1 24.9801,E2 353.0852} C_DIS
LIN {X -11.3307,Y 112.3097,Z 114,A 90.9238,B 24.9332,C -1.8872,E1 24.9852,E2 354.9292} C_DIS
LIN {X -7.7885,Y 112.6101,Z 114,A 89.0366,B 24.9334,C -1.8846,E1 24.9904,E2 356.8235} C_DIS
LIN {X -4.3265,Y 112.7972,Z 114,A 86.6539,B 24.9352,C -1.8594,E1 24.9973,E2 359.2664} C_DIS
LIN {X 0.1639,Y 112.8801,Z 114,A 85.1626,B 24.9329,C -1.8926,E1 25.0012,E2 360.679} C_DIS
LIN {X 3.5365,Y 112.8236,Z 114,A 83.2294,B 24.9335,C -1.8836,E1 25.0067,E2 362.6333} C_DIS
LIN {X 7.5237,Y 112.628,Z 114,A 81.2809,B 24.9333,C -1.8868,E1 25.0121,E2 364.5732} C_DIS
LIN {X 11.3201,Y 112.3108,Z 114,A 79.2904,B 24.9334,C -1.8842,E1 25.0176,E2 366.5688} C_DIS
LIN {X 15.0006,Y 111.8789,Z 114,A 77.3457,B 24.9337,C -1.8812,E1 25.023,E2 368.5192} C_DIS
LIN {X 18.6613,Y 111.3257,Z 114,A 75.5653,B 24.9334,C -1.8847,E1 25.0279,E2 370.2894} C_DIS
LIN {X 22.3547,Y 110.6438,Z 114,A 73.6436,B 24.9335,C -1.8833,E1 25.0332,E2 372.2122} C_DIS
LIN {X 26.1438,Y 109.8115,Z 114,A 71.693,B 24.9335,C -1.883,E1 25.0385,E2 374.1608} C_DIS
LIN {X 29.0077,Y 109.089,Z 114,A 70.1315,B 24.9338,C -1.8794,E1 25.0427,E2 375.7284} C_DIS
LIN {X 32.6661,Y 108.0506,Z 114,A 68.2461,B 24.9338,C -1.8799,E1 25.0478,E2 377.6093} C_DIS
LIN {X 35.9809,Y 106.9909,Z 114,A 66.6608,B 24.9333,C -1.8863,E1 25.0519,E2 379.1766} C_DIS
LIN {X 38.6882,Y 106.0419,Z 114,A 65.0718,B 24.9338,C -1.8792,E1 25.0561,E2 380.7791} C_DIS
LIN {X 41.3218,Y 105.0437,Z 114,A 63.5133,B 24.9343,C -1.8723,E1 25.0602,E2 382.3506} C_DIS
LIN {X 45.0479,Y 103.5005,Z 114,A 61.6649,B 24.9338,C -1.8786,E1 25.0649,E2 384.1796} C_DIS
LIN {X 47.4567,Y 102.4186,Z 114,A 60.3371,B 24.9339,C -1.8776,E1 25.0683,E2 385.5065} C_DIS
LIN {X 49.8978,Y 101.2519,Z 114,A 59.0395,B 24.9339,C -1.8792,E1 25.0715,E2 386.7969} C_DIS
LIN {X 52.5576,Y 99.8968,Z 114,A 57.4195,B 24.9343,C -1.8727,E1 25.0756,E2 388.4279} C_DIS
LIN {X 55.7618,Y 98.1458,Z 114,A 55.4473,B 24.9348,C -1.8649,E1 25.0804,E2 390.4128} C_DIS
LIN {X 58.2942,Y 96.6623,Z 114,A 54.0533,B 24.9347,C -1.8668,E1 25.0837,E2 391.7978} C_DIS
LIN {X 61.5708,Y 94.6105,Z 114,A 51.97,B 24.9353,C -1.8584,E1 25.0887,E2 393.8943} C_DIS
LIN {X 64.2219,Y 92.8293,Z 114,A 50.6428,B 24.9345,C -1.8686,E1 25.0917,E2 395.1928} C_DIS
LIN {X 66.6088,Y 91.1315,Z 114,A 49.01,B 24.9352,C -1.8596,E1 25.0954,E2 396.8411} C_DIS
LIN {X 68.8841,Y 89.424,Z 114,A 47.6156,B 24.9352,C -1.8592,E1 25.0985,E2 398.2315} C_DIS
LIN {X 72.6785,Y 86.3711,Z 114,A 45.0437,B 24.9358,C -1.8501,E1 25.1041,E2 400.8152} C_DIS
LIN {X 74.9608,Y 84.3963,Z 114,A 43.4938,B 24.9361,C -1.8462,E1 25.1073,E2 402.3681} C_DIS
LIN {X 77.102,Y 82.4442,Z 114,A 41.9383,B 24.9366,C -1.8395,E1 25.1106,E2 403.9332} C_DIS
LIN {X 80.1223,Y 79.5119,Z 114,A 40.0263,B 24.9362,C -1.8448,E1 25.1143,E2 405.8244} C_DIS
LIN {X 84.6496,Y 74.6754,Z 114,A 36.6939,B 24.9366,C -1.8386,E1 25.1206,E2 409.157} C_DIS
LIN {X 86.4127,Y 72.6286,Z 114,A 35.1313,B 24.9374,C -1.8268,E1 25.1235,E2 410.7402} C_DIS
LIN {X 89.9831,Y 68.1535,Z 114,A 32.4326,B 24.9373,C -1.829,E1 25.1281,E2 413.421} C_DIS
LIN {X 91.5303,Y 66.0625,Z 114,A 30.9544,B 24.938,C -1.8186,E1 25.1306,E2 414.9166} C_DIS
LIN {X 93.8881,Y 62.6665,Z 114,A 28.9772,B 24.938,C -1.8186,E1 25.1337,E2 416.8839} C_DIS
LIN {X 95.4851,Y 60.2036,Z 114,A 27.4423,B 24.9384,C -1.8128,E1 25.136,E2 418.425} C_DIS
LIN {X 97.4446,Y 56.978,Z 114,A 25.5211,B 24.9388,C -1.8074,E1 25.1387,E2 420.3492} C_DIS
LIN {X 98.8798,Y 54.451,Z 114,A 24.0252,B 24.9391,C -1.8024,E1 25.1408,E2 421.849} C_DIS
LIN {X 100.5297,Y 51.3365,Z 114,A 22.3438,B 24.9391,C -1.8023,E1 25.1429,E2 423.5218} C_DIS
LIN {X 102.2491,Y 47.8208,Z 114,A 20.3471,B 24.9395,C -1.7962,E1 25.1453,E2 425.5221} C_DIS
LIN {X 103.8455,Y 44.2491,Z 114,A 18.2136,B 24.9404,C -1.7837,E1 25.1477,E2 427.6733} C_DIS
LIN {X 105.517,Y 40.0978,Z 114,A 16.1498,B 24.9402,C -1.7865,E1 25.1498,E2 429.7192} C_DIS
LIN {X 106.8157,Y 36.5004,Z 114,A 14.3824,B 24.94,C -1.7886,E1 25.1514,E2 431.4717} C_DIS
LIN {X 107.6945,Y 33.8191,Z 114,A 12.7761,B 24.9409,C -1.7763,E1 25.1528,E2 433.0979} C_DIS
LIN {X 108.7861,Y 30.1279,Z 114,A 10.7433,B 24.9415,C -1.7667,E1 25.1544,E2 435.1417} C_DIS
LIN {X 109.6735,Y 26.7096,Z 114,A 9.0236,B 24.9416,C -1.7645,E1 25.1556,E2 436.8567} C_DIS
LIN {X 110.5552,Y 22.7866,Z 114,A 7.2399,B 24.9413,C -1.7698,E1 25.1566,E2 438.6174} C_DIS
LIN {X 111.1019,Y 19.9506,Z 114,A 5.666,B 24.9419,C -1.7603,E1 25.1574,E2 440.2046} C_DIS
LIN {X 111.6398,Y 16.6895,Z 114,A 3.819,B 24.9428,C -1.7472,E1 25.1582,E2 442.0716} C_DIS
LIN {X 112.0848,Y 13.3688,Z 114,A 2.4136,B 24.9423,C -1.7553,E1 25.1587,E2 443.4497} C_DIS
LIN {X 112.3436,Y 10.9985,Z 114,A 0.9412,B 24.9433,C -1.7393,E1 25.1592,E2 444.9509} C_DIS
LIN {X 112.6276,Y 7.5293,Z 114,A -0.6831,B 24.9433,C -1.7402,E1 25.1595,E2 446.5635} C_DIS
LIN {X 112.7686,Y 4.9938,Z 114,A -2.1589,B 24.9441,C -1.7275,E1 25.1597,E2 448.0606} C_DIS
LIN {X 112.8206,Y -3.6352,Z 114,A -6.1372,B 24.9438,C -1.7316,E1 25.1597,E2 452.0054} C_DIS
LIN {X 112.4775,Y -9.5266,Z 114,A -9.9113,B 24.9467,C -1.6862,E1 25.1589,E2 455.8641} C_DIS
LIN {X 112.0362,Y -13.7832,Z 114,A -11.6144,B 24.9458,C -1.7005,E1 25.1584,E2 457.5234} C_DIS
LIN {X 111.5188,Y -17.4721,Z 114,A -13.3272,B 24.9457,C -1.7026,E1 25.1577,E2 459.2214} C_DIS
LIN {X 110.8908,Y -21.0938,Z 114,A -15.1895,B 24.9461,C -1.6967,E1 25.1568,E2 461.0866} C_DIS
LIN {X 110.2263,Y -24.3291,Z 114,A -16.9884,B 24.9468,C -1.6857,E1 25.1557,E2 462.9011} C_DIS
LIN {X 109.2831,Y -28.2647,Z 114,A -18.9478,B 24.9468,C -1.6834,E1 25.1544,E2 464.8544} C_DIS
LIN {X 108.2581,Y -31.9667,Z 114,A -20.6764,B 24.9466,C -1.6874,E1 25.1531,E2 466.5638} C_DIS
LIN {X 107.3918,Y -34.766,Z 114,A -22.3381,B 24.9474,C -1.6746,E1 25.1517,E2 468.2461} C_DIS
LIN {X 106.1192,Y -38.4763,Z 114,A -24.2962,B 24.9477,C -1.6699,E1 25.1499,E2 470.2043} C_DIS
LIN {X 104.8873,Y -41.7198,Z 114,A -25.9899,B 24.9479,C -1.6675,E1 25.1482,E2 471.8943} C_DIS
LIN {X 103.4597,Y -45.1416,Z 114,A -27.8086,B 24.9481,C -1.6646,E1 25.1462,E2 473.7099} C_DIS
LIN {X 102.0433,Y -48.2629,Z 114,A -29.9116,B 24.9494,C -1.6427,E1 25.1437,E2 475.8532} C_DIS
LIN {X 99.9317,Y -52.4914,Z 114,A -32.0664,B 24.9492,C -1.6467,E1 25.141,E2 477.9872} C_DIS
LIN {X 98.1812,Y -55.7001,Z 114,A -34.0075,B 24.9498,C -1.6372,E1 25.1383,E2 479.9403} C_DIS
LIN {X 96.3322,Y -58.8374,Z 114,A -35.7469,B 24.9498,C -1.6369,E1 25.1358,E2 481.6717} C_DIS
LIN {X 94.7621,Y -61.335,Z 114,A -37.3516,B 24.9504,C -1.6277,E1 25.1334,E2 483.2899} C_DIS
LIN {X 92.6879,Y -64.4253,Z 114,A -39.1175,B 24.9504,C -1.628,E1 25.1306,E2 485.0465} C_DIS
LIN {X 90.6788,Y -67.227,Z 114,A -41.0108,B 24.951,C -1.6166,E1 25.1275,E2 486.9575} C_DIS
LIN {X 88.0252,Y -70.6647,Z 114,A -43.0845,B 24.951,C -1.6166,E1 25.1239,E2 489.0215} C_DIS
LIN {X 85.8747,Y -73.2613,Z 114,A -44.7157,B 24.951,C -1.6158,E1 25.121,E2 490.6472} C_DIS
LIN {X 83.4936,Y -75.9652,Z 114,A -46.3889,B 24.951,C -1.6181,E1 25.1179,E2 492.3075} C_DIS
LIN {X 81.7316,Y -77.8591,Z 114,A -47.9502,B 24.9518,C -1.6035,E1 25.1149,E2 493.8963} C_DIS
LIN {X 79.1651,Y -80.4649,Z 114,A -49.7547,B 24.952,C -1.6013,E1 25.1113,E2 495.6983} C_DIS
LIN {X 76.4977,Y -83.005,Z 114,A -51.426,B 24.9517,C -1.6058,E1 25.1079,E2 497.3523} C_DIS
LIN {X 74.6163,Y -84.7013,Z 114,A -52.885,B 24.9523,C -1.595,E1 25.1048,E2 498.831} C_DIS
LIN {X 72.1025,Y -86.8499,Z 114,A -54.5899,B 24.9526,C -1.59,E1 25.1012,E2 500.541} C_DIS
LIN {X 69.0999,Y -89.2577,Z 114,A -56.5564,B 24.9529,C -1.5851,E1 25.0969,E2 502.5117} C_DIS
LIN {X 66.0662,Y -91.5276,Z 114,A -58.4822,B 24.9532,C -1.581,E1 25.0925,E2 504.4406} C_DIS
LIN {X 62.9613,Y -93.6893,Z 114,A -60.3599,B 24.9532,C -1.579,E1 25.0882,E2 506.3166} C_DIS
LIN {X 60.2598,Y -95.4501,Z 114,A -61.7633,B 24.9529,C -1.5862,E1 25.0849,E2 507.6983} C_DIS
LIN {X 58.1122,Y -96.7729,Z 114,A -63.3128,B 24.9537,C -1.5718,E1 25.0812,E2 509.277} C_DIS
LIN {X 54.8362,Y -98.6646,Z 114,A -65.1172,B 24.9537,C -1.5735,E1 25.0768,E2 511.0721} C_DIS
LIN {X 51.3426,Y -100.5266,Z 114,A -67.1464,B 24.9539,C -1.5692,E1 25.0718,E2 513.1058} C_DIS
LIN {X 48.7299,Y -101.8189,Z 114,A -68.6798,B 24.9541,C -1.5644,E1 25.0679,E2 514.6465} C_DIS
LIN {X 45.0479,Y -103.5005,Z 114,A -70.7486,B 24.9544,C -1.5606,E1 25.0626,E2 516.7191} C_DIS
LIN {X 41.8593,Y -104.8326,Z 114,A -72.4712,B 24.9544,C -1.5594,E1 25.0582,E2 518.4406} C_DIS
LIN {X 38.4798,Y -106.1179,Z 114,A -74.2,B 24.9544,C -1.5617,E1 25.0537,E2 520.1605} C_DIS
LIN {X 35.3789,Y -107.1935,Z 114,A -75.9585,B 24.9547,C -1.5555,E1 25.049,E2 521.9302} C_DIS
LIN {X 32.4969,Y -108.1008,Z 114,A -77.1969,B 24.954,C -1.5667,E1 25.0458,E2 523.1399} C_DIS
LIN {X 29.5183,Y -108.9511,Z 114,A -78.998,B 24.9547,C -1.5549,E1 25.0408,E2 524.9659} C_DIS
LIN {X 25.7242,Y -109.9092,Z 114,A -80.9051,B 24.9547,C -1.5564,E1 25.0357,E2 526.8667} C_DIS
LIN {X 23.2097,Y -110.4683,Z 114,A -82.1485,B 24.9545,C -1.558,E1 25.0323,E2 528.1047} C_DIS
LIN {X 20.0439,Y -111.0852,Z 114,A -83.9264,B 24.955,C -1.5505,E1 25.0274,E2 529.8982} C_DIS
LIN {X 16.0857,Y -111.7272,Z 114,A -85.9226,B 24.955,C -1.5507,E1 25.0219,E2 531.892} C_DIS
LIN {X 13.3019,Y -112.0926,Z 114,A -88.0404,B 24.9567,C -1.5201,E1 25.0158,E2 534.0809} C_DIS
LIN {X 8.5192,Y -112.5581,Z 114,A -89.8193,B 24.9552,C -1.5471,E1 25.011,E2 535.7947} C_DIS
LIN {X 4.8531,Y -112.7746,Z 114,A -91.6747,B 24.9552,C -1.5468,E1 25.0059,E2 537.6503} C_DIS
LIN {X 0.7919,Y -112.8763,Z 114,A -92.9036,B 24.9531,C -1.5821,E1 25.0027,E2 538.7952} C_DIS
Enddeposition()
LIN {X 0.7919,Y -112.8763,Z 114,A -92.9036,B 24.9531,C -1.5821,E1 25.0027,E2 538.7952} C_DIS
Startdeposition()
$VEL.CP = VEL_PRINT
LIN {X 2.3682,Y -111.9354,Z 114,A -92.2423,B 24.9525,C -1.5919,E1 25.0046,E2 538.1108} C_DIS
LIN {X 5.9698,Y -111.801,Z 114,A -90.2558,B 24.9521,C -1.5988,E1 25.0102,E2 536.1087} C_DIS
LIN {X 10.5813,Y -111.4593,Z 114,A -87.726,B 24.9516,C -1.6071,E1 25.0173,E2 533.5606} C_DIS
LIN {X 14.8024,Y -110.978,Z 114,A -85.6542,B 24.9518,C -1.604,E1 25.023,E2 531.4978} C_DIS
LIN {X 18.4982,Y -110.4214,Z 114,A -83.8462,B 24.952,C -1.6008,E1 25.0279,E2 529.699} C_DIS
LIN {X 22.3519,Y -109.7063,Z 114,A -81.8608,B 24.952,C -1.6016,E1 25.0334,E2 527.714} C_DIS
LIN {X 25.439,Y -109.032,Z 114,A -80.15,B 24.9516,C -1.6073,E1 25.0381,E2 525.9922} C_DIS
LIN {X 30.6549,Y -107.6817,Z 114,A -77.4721,B 24.9516,C -1.6067,E1 25.0453,E2 523.3198} C_DIS
LIN {X 34.0805,Y -106.6478,Z 114,A -75.5491,B 24.9513,C -1.6129,E1 25.0504,E2 521.3856} C_DIS
LIN {X 37.6449,Y -105.4433,Z 114,A -73.6688,B 24.9513,C -1.6134,E1 25.0554,E2 519.508} C_DIS
LIN {X 40.9246,Y -104.2125,Z 114,A -71.3353,B 24.9496,C -1.64,E1 25.0616,E2 517.1166} C_DIS
LIN {X 44.9313,Y -102.5489,Z 114,A -69.8818,B 24.9515,C -1.6091,E1 25.0651,E2 515.7397} C_DIS
LIN {X 47.3615,Y -101.4493,Z 114,A -68.0629,B 24.9501,C -1.6315,E1 25.0699,E2 513.8725} C_DIS
LIN {X 51.6955,Y -99.3122,Z 114,A -65.8299,B 24.9505,C -1.6249,E1 25.0754,E2 511.6612} C_DIS
LIN {X 54.7999,Y -97.6324,Z 114,A -64.1383,B 24.9506,C -1.623,E1 25.0795,E2 509.9792} C_DIS
LIN {X 59.3813,Y -94.9154,Z 114,A -61.4101,B 24.9503,C -1.6282,E1 25.086,E2 507.2471} C_DIS
LIN {X 61.6329,Y -93.469,Z 114,A -60.0508,B 24.9502,C -1.6304,E1 25.0892,E2 505.887} C_DIS
LIN {X 64.7175,Y -91.3611,Z 114,A -58.0726,B 24.9498,C -1.6373,E1 25.0937,E2 503.8993} C_DIS
LIN {X 67.8997,Y -89.0224,Z 114,A -55.9592,B 24.9492,C -1.6458,E1 25.0985,E2 501.7735} C_DIS
LIN {X 70.5634,Y -86.9245,Z 114,A -54.386,B 24.9495,C -1.6423,E1 25.1019,E2 500.2145} C_DIS
LIN {X 73.5496,Y -84.4129,Z 114,A -52.4145,B 24.9492,C -1.6457,E1 25.1061,E2 498.2425} C_DIS
LIN {X 75.7974,Y -82.4004,Z 114,A -50.8887,B 24.9491,C -1.6485,E1 25.1092,E2 496.7163} C_DIS
LIN {X 78.4375,Y -79.892,Z 114,A -48.9824,B 24.9487,C -1.655,E1 25.1131,E2 494.8027} C_DIS
LIN {X 81.047,Y -77.2453,Z 114,A -47.0064,B 24.9482,C -1.6631,E1 25.1169,E2 492.8161} C_DIS
LIN {X 83.5681,Y -74.5082,Z 114,A -45.258,B 24.9483,C -1.6609,E1 25.1202,E2 491.0806} C_DIS
LIN {X 85.9173,Y -71.7869,Z 114,A -43.391,B 24.9479,C -1.6669,E1 25.1236,E2 489.2078} C_DIS
LIN {X 88.0826,Y -69.1134,Z 114,A -41.7056,B 24.9479,C -1.6682,E1 25.1265,E2 487.5273} C_DIS
LIN {X 89.7646,Y -66.9144,Z 114,A -40.2219,B 24.9474,C -1.6751,E1 25.129,E2 486.0343} C_DIS
LIN {X 91.7418,Y -64.1764,Z 114,A -38.3063,B 24.9466,C -1.6885,E1 25.1321,E2 484.0964} C_DIS
LIN {X 95.782,Y -57.9734,Z 114,A -34.8298,B 24.9468,C -1.685,E1 25.1373,E2 480.6456} C_DIS
LIN {X 97.149,Y -55.652,Z 114,A -33.4321,B 24.9465,C -1.6899,E1 25.1393,E2 479.2436} C_DIS
LIN {X 98.606,Y -53.029,Z 114,A -30.9242,B 24.9433,C -1.7395,E1 25.1427,E2 476.6321} C_DIS
LIN {X 101.2126,Y -47.87,Z 114,A -28.9886,B 24.9458,C -1.701,E1 25.145,E2 474.7976} C_DIS
LIN {X 102.8822,Y -44.1668,Z 114,A -26.5055,B 24.9442,C -1.726,E1 25.1478,E2 472.2691} C_DIS
LIN {X 104.3565,Y -40.558,Z 114,A -24.7785,B 24.9446,C -1.7198,E1 25.1495,E2 470.5663} C_DIS
LIN {X 105.6775,Y -36.9776,Z 114,A -22.9244,B 24.9445,C -1.7214,E1 25.1513,E2 468.7188} C_DIS
LIN {X 106.903,Y -33.2688,Z 114,A -20.5691,B 24.943,C -1.7442,E1 25.1533,E2 466.3232} C_DIS
LIN {X 107.8618,Y -30.0193,Z 114,A -19.2884,B 24.944,C -1.7288,E1 25.1542,E2 465.0862} C_DIS
LIN {X 108.8243,Y -26.3132,Z 114,A -17.2095,B 24.9432,C -1.7406,E1 25.1557,E2 462.9914} C_DIS
LIN {X 109.6901,Y -22.4307,Z 114,A -15.2427,B 24.943,C -1.744,E1 25.1568,E2 461.0281} C_DIS
LIN {X 110.4104,Y -18.5637,Z 114,A -13.2474,B 24.9426,C -1.7497,E1 25.1578,E2 459.031} C_DIS
LIN {X 110.9696,Y -14.8673,Z 114,A -11.2962,B 24.9421,C -1.7576,E1 25.1586,E2 457.0726} C_DIS
LIN {X 111.4545,Y -10.6334,Z 114,A -8.9216,B 24.941,C -1.7737,E1 25.1592,E2 454.6741} C_DIS
LIN {X 111.8617,Y -4.694,Z 114,A -6.1578,B 24.9412,C -1.7705,E1 25.1597,E2 451.9342} C_DIS
LIN {X 111.938,Y 2.2282,Z 114,A -2.5459,B 24.9403,C -1.7852,E1 25.1597,E2 448.3092} C_DIS
LIN {X 111.8003,Y 5.9829,Z 114,A -0.719,B 24.9401,C -1.787,E1 25.1595,E2 446.4889} C_DIS
LIN {X 111.5459,Y 9.6436,Z 114,A 1.2545,B 24.9394,C -1.7974,E1 25.159,E2 444.5026} C_DIS
LIN {X 111.1653,Y 13.3198,Z 114,A 3.1111,B 24.9391,C -1.8019,E1 25.1585,E2 442.6463} C_DIS
LIN {X 110.6355,Y 17.171,Z 114,A 4.9456,B 24.9391,C -1.8011,E1 25.1577,E2 440.8245} C_DIS
LIN {X 110.0567,Y 20.5657,Z 114,A 6.8425,B 24.9384,C -1.8128,E1 25.1568,E2 438.911} C_DIS
LIN {X 109.245,Y 24.5161,Z 114,A 8.8987,B 24.938,C -1.8189,E1 25.1556,E2 436.8525} C_DIS
LIN {X 108.3748,Y 28.1071,Z 114,A 10.6595,B 24.938,C -1.8189,E1 25.1544,E2 435.102} C_DIS
LIN {X 106.7496,Y 33.7638,Z 114,A 13.7019,B 24.9373,C -1.8294,E1 25.152,E2 432.0521} C_DIS
LIN {X 105.6645,Y 37.0145,Z 114,A 15.4273,B 24.937,C -1.8334,E1 25.1504,E2 430.327} C_DIS
LIN {X 103.1601,Y 43.5091,Z 114,A 18.9071,B 24.9365,C -1.8401,E1 25.1468,E2 426.8507} C_DIS
LIN {X 101.9087,Y 46.3664,Z 114,A 20.6276,B 24.9358,C -1.8503,E1 25.1448,E2 425.1154} C_DIS
LIN {X 100.3269,Y 49.6948,Z 114,A 22.3871,B 24.9358,C -1.8499,E1 25.1427,E2 423.3663} C_DIS
LIN {X 98.8457,Y 52.5814,Z 114,A 24.2881,B 24.9348,C -1.8655,E1 25.1402,E2 421.4387} C_DIS
LIN {X 97.0279,Y 55.8628,Z 114,A 25.9648,B 24.9352,C -1.8597,E1 25.1379,E2 419.7843} C_DIS
LIN {X 94.8259,Y 59.5245,Z 114,A 28.0492,B 24.9351,C -1.8609,E1 25.1349,E2 417.7077} C_DIS
LIN {X 93.2405,Y 61.9793,Z 114,A 29.7224,B 24.9343,C -1.8728,E1 25.1323,E2 416.0148} C_DIS
LIN {X 91.1519,Y 65.0106,Z 114,A 31.5022,B 24.9343,C -1.8728,E1 25.1295,E2 414.2434} C_DIS
LIN {X 89.4,Y 67.3998,Z 114,A 33.2679,B 24.9332,C -1.8879,E1 25.1265,E2 412.4507} C_DIS
LIN {X 86.7896,Y 70.7299,Z 114,A 35.0549,B 24.934,C -1.8761,E1 25.1234,E2 410.7} C_DIS
LIN {X 85.0029,Y 72.8676,Z 114,A 36.6154,B 24.9334,C -1.8854,E1 25.1206,E2 409.1244} C_DIS
LIN {X 80.3492,Y 77.9691,Z 114,A 40.0376,B 24.9332,C -1.8883,E1 25.1141,E2 405.7105} C_DIS
LIN {X 77.558,Y 80.7456,Z 114,A 42.2273,B 24.9323,C -1.9004,E1 25.1097,E2 403.5014} C_DIS
LIN {X 74.6111,Y 83.476,Z 114,A 44.1132,B 24.9325,C -1.897,E1 25.1058,E2 401.631} C_DIS
LIN {X 72.2882,Y 85.4965,Z 114,A 45.8767,B 24.9317,C -1.9085,E1 25.102,E2 399.8475} C_DIS
LIN {X 69.2959,Y 87.9384,Z 114,A 47.701,B 24.9319,C -1.9054,E1 25.0981,E2 398.0372} C_DIS
LIN {X 66.0962,Y 90.3679,Z 114,A 49.6977,B 24.9319,C -1.9065,E1 25.0936,E2 396.0452} C_DIS
LIN {X 63.3085,Y 92.3445,Z 114,A 51.4958,B 24.9315,C -1.9116,E1 25.0895,E2 394.2412} C_DIS
LIN {X 59.5245,Y 94.8259,Z 114,A 53.534,B 24.9321,C -1.9031,E1 25.0848,E2 392.2297} C_DIS
LIN {X 56.5515,Y 96.6293,Z 114,A 55.5274,B 24.9312,C -1.9151,E1 25.0799,E2 390.2141} C_DIS
LIN {X 53.014,Y 98.6142,Z 114,A 57.5271,B 24.9312,C -1.9147,E1 25.0751,E2 388.2212} C_DIS
LIN {X 50.7647,Y 99.79,Z 114,A 58.8434,B 24.9311,C -1.9171,E1 25.0718,E2 386.9027} C_DIS
LIN {X 48.1986,Y 101.0547,Z 114,A 60.461,B 24.9305,C -1.9256,E1 25.0677,E2 385.2693} C_DIS
LIN {X 44.7364,Y 102.6339,Z 114,A 62.2696,B 24.9308,C -1.9218,E1 25.0631,E2 383.4741} C_DIS
LIN {X 41.6994,Y 103.9063,Z 114,A 64.21,B 24.9298,C -1.9346,E1 25.058,E2 381.5079} C_DIS
LIN {X 37.8068,Y 105.3853,Z 114,A 66.0443,B 24.9306,C -1.9238,E1 25.0533,E2 379.7032} C_DIS
LIN {X 34.9389,Y 106.37,Z 114,A 67.7181,B 24.9301,C -1.9304,E1 25.0488,E2 378.017} C_DIS
LIN {X 30.1533,Y 107.8238,Z 114,A 70.1787,B 24.9303,C -1.928,E1 25.0423,E2 375.5663} C_DIS
LIN {X 26.2625,Y 108.8366,Z 114,A 72.3702,B 24.9298,C -1.935,E1 25.0363,E2 373.3616} C_DIS
LIN {X 22.4977,Y 109.6764,Z 114,A 74.2191,B 24.9301,C -1.9306,E1 25.0313,E2 371.5254} C_DIS
LIN {X 19.3871,Y 110.2696,Z 114,A 75.9815,B 24.9296,C -1.9372,E1 25.0264,E2 369.7492} C_DIS
LIN {X 15.7567,Y 110.8458,Z 114,A 77.7345,B 24.93,C -1.9323,E1 25.0216,E2 368.0094} C_DIS
LIN {X 12.2691,Y 111.2875,Z 114,A 79.6467,B 24.9296,C -1.9375,E1 25.0163,E2 366.0865} C_DIS
LIN {X 8.7258,Y 111.6197,Z 114,A 81.3165,B 24.9301,C -1.9312,E1 25.0117,E2 364.4323} C_DIS
LIN {X 5.3471,Y 111.8336,Z 114,A 83.1841,B 24.9297,C -1.9369,E1 25.0064,E2 362.5521} C_DIS
LIN {X 1.8663,Y 111.9447,Z 114,A 84.8693,B 24.93,C -1.9326,E1 25.0018,E2 360.8774} C_DIS
LIN {X -2.6145,Y 111.9306,Z 114,A 87.4057,B 24.9293,C -1.9423,E1 24.9946,E2 358.3179} C_DIS
LIN {X -7.2558,Y 111.7251,Z 114,A 89.6163,B 24.9298,C -1.9344,E1 24.9885,E2 356.1253} C_DIS
LIN {X -10.4671,Y 111.4699,Z 114,A 91.151,B 24.9302,C -1.9289,E1 24.9843,E2 354.6031} C_DIS
LIN {X -13.3368,Y 111.1633,Z 114,A 92.6628,B 24.9302,C -1.9295,E1 24.9801,E2 353.0888} C_DIS
LIN {X -16.8652,Y 110.6828,Z 114,A 94.5383,B 24.9302,C -1.9305,E1 24.9749,E2 351.2094} C_DIS
LIN {X -20.6953,Y 110.0318,Z 114,A 96.5768,B 24.9301,C -1.931,E1 24.9693,E2 349.1675} C_DIS
LIN {X -24.2074,Y 109.3123,Z 114,A 98.296,B 24.9306,C -1.9247,E1 24.9646,E2 347.4612} C_DIS
LIN {X -27.5898,Y 108.5078,Z 114,A 100.4248,B 24.9296,C -1.9374,E1 24.9587,E2 345.2993} C_DIS
LIN {X -31.776,Y 107.3562,Z 114,A 103.2549,B 24.928,C -1.9601,E1 24.951,E2 342.4105} C_DIS
LIN {X -37.0156,Y 105.6641,Z 114,A 104.8239,B 24.9319,C -1.9053,E1 24.9472,E2 340.9688} C_DIS
LIN {X -39.4768,Y 104.7696,Z 114,A 107.4494,B 24.9283,C -1.9562,E1 24.94,E2 338.2169} C_DIS
LIN {X -44.672,Y 102.6619,Z 114,A 109.1053,B 24.9322,C -1.9024,E1 24.9361,E2 336.6851} C_DIS
LIN {X -47.1844,Y 101.5318,Z 114,A 110.8505,B 24.9313,C -1.9138,E1 24.9315,E2 334.9084} C_DIS
LIN {X -50.9436,Y 99.6986,Z 114,A 113.1672,B 24.9311,C -1.9175,E1 24.9257,E2 332.5769} C_DIS
LIN {X -55.6699,Y 97.1387,Z 114,A 115.7254,B 24.932,C -1.9049,E1 24.9195,E2 330.0412} C_DIS
LIN {X -58.6068,Y 95.397,Z 114,A 118.0066,B 24.9307,C -1.9232,E1 24.914,E2 327.7094} C_DIS
LIN {X -61.8408,Y 93.3318,Z 114,A 119.5725,B 24.9321,C -1.9033,E1 24.9104,E2 326.1857} C_DIS
LIN {X -64.9651,Y 91.1845,Z 114,A 121.4033,B 24.9327,C -1.895,E1 24.9063,E2 324.3684} C_DIS
LIN {X -67.415,Y 89.3886,Z 114,A 123.4378,B 24.9315,C -1.911,E1 24.9016,E2 322.2885} C_DIS
LIN {X -70.315,Y 87.1258,Z 114,A 125.0242,B 24.9327,C -1.895,E1 24.8982,E2 320.7343} C_DIS
LIN {X -72.8304,Y 85.0346,Z 114,A 126.5769,B 24.9333,C -1.8864,E1 24.895,E2 319.196} C_DIS
LIN {X -75.5214,Y 82.6537,Z 114,A 128.4589,B 24.9335,C -1.8839,E1 24.891,E2 317.3126} C_DIS
LIN {X -79.1215,Y 79.216,Z 114,A 131.2941,B 24.9331,C -1.8892,E1 24.8853,E2 314.4529} C_DIS
LIN {X -82.666,Y 75.5079,Z 114,A 133.5267,B 24.9347,C -1.867,E1 24.8812,E2 312.2632} C_DIS
LIN {X -84.8585,Y 73.037,Z 114,A 135.7364,B 24.9335,C -1.8832,E1 24.877,E2 310.0049} C_DIS
LIN {X -87.0939,Y 70.3543,Z 114,A 138.0302,B 24.9324,C -1.8987,E1 24.873,E2 307.6634} C_DIS
LIN {X -90.5744,Y 65.8141,Z 114,A 139.947,B 24.9358,C -1.8506,E1 24.8699,E2 305.8521} C_DIS
LIN {X -92.4562,Y 63.1436,Z 114,A 143.098,B 24.932,C -1.9047,E1 24.8648,E2 302.5564} C_DIS
LIN {X -96.5073,Y 56.7579,Z 114,A 145.5054,B 24.9369,C -1.8355,E1 24.8615,E2 300.3018} C_DIS
LIN {X -97.86,Y 54.3924,Z 114,A 146.9866,B 24.9369,C -1.8348,E1 24.8595,E2 298.8145} C_DIS
LIN {X -99.6281,Y 51.0816,Z 114,A 148.9818,B 24.9371,C -1.832,E1 24.8569,E2 296.8153} C_DIS
LIN {X -101.268,Y 47.7511,Z 114,A 150.887,B 24.9375,C -1.8265,E1 24.8546,E2 294.9129} C_DIS
LIN {X -103.2449,Y 43.3079,Z 114,A 153.423,B 24.9379,C -1.8207,E1 24.8518,E2 292.3766} C_DIS
LIN {X -104.9,Y 39.1326,Z 114,A 155.767,B 24.9382,C -1.8154,E1 24.8494,E2 290.0322} C_DIS
LIN {X -106.1247,Y 35.6737,Z 114,A 158.4571,B 24.9364,C -1.8414,E1 24.847,E2 287.2646} C_DIS
LIN {X -107.738,Y 30.4563,Z 114,A 161.099,B 24.9375,C -1.8265,E1 24.845,E2 284.643} C_DIS
LIN {X -108.9473,Y 25.8058,Z 114,A 162.76,B 24.9401,C -1.7873,E1 24.8439,E2 283.0658} C_DIS
LIN {X -109.5978,Y 22.8806,Z 114,A 164.8684,B 24.9389,C -1.8049,E1 24.8427,E2 280.9031} C_DIS
LIN {X -110.2962,Y 19.2394,Z 114,A 166.3372,B 24.9405,C -1.782,E1 24.842,E2 279.4803} C_DIS
LIN {X -110.8525,Y 15.7091,Z 114,A 168.1372,B 24.941,C -1.7749,E1 24.8412,E2 277.6862} C_DIS
LIN {X -111.2359,Y 12.717,Z 114,A 169.6691,B 24.9413,C -1.7695,E1 24.8407,E2 276.1582} C_DIS
LIN {X -111.5417,Y 9.6892,Z 114,A 171.5426,B 24.9408,C -1.7767,E1 24.8402,E2 274.2562} C_DIS
LIN {X -111.8139,Y 5.7371,Z 114,A 173.5697,B 24.9413,C -1.7701,E1 24.8399,E2 272.2326} C_DIS
LIN {X -111.9565,Y 0.9833,Z 114,A 175.8058,B 24.9423,C -1.7545,E1 24.8398,E2 270.0203} C_DIS
LIN {X -111.9254,Y -2.8484,Z 114,A 177.9619,B 24.9423,C -1.7558,E1 24.8398,E2 267.8482} C_DIS
LIN {X -111.7203,Y -7.3268,Z 114,A -179.9461,B 24.9432,C -1.7405,E1 24.8402,E2 265.7801} C_DIS
LIN {X -111.4825,Y -10.3305,Z 114,A -178.4164,B 24.9436,C -1.735,E1 24.8406,E2 264.2541} C_DIS
LIN {X -111.1141,Y -13.752,Z 114,A -176.4609,B 24.9435,C -1.737,E1 24.8412,E2 262.2823} C_DIS
LIN {X -110.4784,Y -18.1569,Z 114,A -174.5682,B 24.9449,C -1.7147,E1 24.842,E2 260.4313} C_DIS
LIN {X -109.7328,Y -22.2229,Z 114,A -172.1134,B 24.9445,C -1.7213,E1 24.8433,E2 257.9463} C_DIS
LIN {X -108.5199,Y -27.5427,Z 114,A -169.614,B 24.9458,C -1.7012,E1 24.8449,E2 255.4803} C_DIS
LIN {X -106.9376,Y -33.1572,Z 114,A -166.3712,B 24.9458,C -1.7021,E1 24.8474,E2 252.2165} C_DIS
LIN {X -105.742,Y -36.7936,Z 114,A -164.3705,B 24.946,C -1.6979,E1 24.8492,E2 250.2146} C_DIS
LIN {X -104.5831,Y -39.9693,Z 114,A -162.5708,B 24.9461,C -1.6955,E1 24.8509,E2 248.4103} C_DIS
LIN {X -103.1794,Y -43.4633,Z 114,A -160.6249,B 24.9464,C -1.6906,E1 24.853,E2 246.4652} C_DIS
LIN {X -101.6133,Y -47.0091,Z 114,A -158.7336,B 24.947,C -1.6813,E1 24.8552,E2 244.5858} C_DIS
LIN {X -100.2347,Y -49.8807,Z 114,A -156.7375,B 24.9464,C -1.6912,E1 24.8577,E2 242.5552} C_DIS
LIN {X -98.7523,Y -52.7569,Z 114,A -155.2508,B 24.9471,C -1.6799,E1 24.8596,E2 241.0877} C_DIS
LIN {X -96.8291,Y -56.2087,Z 114,A -153.2875,B 24.9476,C -1.6721,E1 24.8623,E2 239.1328} C_DIS
LIN {X -94.9647,Y -59.3023,Z 114,A -151.2434,B 24.9474,C -1.675,E1 24.8654,E2 237.0712} C_DIS
LIN {X -92.6365,Y -62.8773,Z 114,A -149.3174,B 24.9484,C -1.6591,E1 24.8683,E2 235.1735} C_DIS
LIN {X -90.4311,Y -66.0098,Z 114,A -146.9853,B 24.9478,C -1.6691,E1 24.8722,E2 232.8062} C_DIS
LIN {X -88.4328,Y -68.6649,Z 114,A -145.7644,B 24.9492,C -1.6457,E1 24.8742,E2 231.6352} C_DIS
LIN {X -86.5479,Y -71.0281,Z 114,A -143.9463,B 24.9488,C -1.6529,E1 24.8774,E2 229.7916} C_DIS
LIN {X -83.9161,Y -74.1183,Z 114,A -141.882,B 24.9491,C -1.6476,E1 24.8812,E2 227.7306} C_DIS
LIN {X -81.4571,Y -76.8103,Z 114,A -140.1372,B 24.9497,C -1.6386,E1 24.8845,E2 225.9996} C_DIS
LIN {X -78.7705,Y -79.563,Z 114,A -138.1387,B 24.9499,C -1.6356,E1 24.8884,E2 223.9998} C_DIS
LIN {X -75.935,Y -82.2742,Z 114,A -136.1194,B 24.9501,C -1.6319,E1 24.8925,E2 221.9809} C_DIS
LIN {X -73.4636,Y -84.4879,Z 114,A -134.4522,B 24.9504,C -1.6273,E1 24.896,E2 220.3181} C_DIS
LIN {X -70.1331,Y -87.2732,Z 114,A -132.0864,B 24.9503,C -1.6289,E1 24.9011,E2 217.9394} C_DIS
LIN {X -67.0597,Y -89.6555,Z 114,A -130.146,B 24.9506,C -1.6234,E1 24.9054,E2 216.0051} C_DIS
LIN {X -62.7859,Y -92.6984,Z 114,A -127.8938,B 24.952,C -1.6012,E1 24.9105,E2 213.798} C_DIS
LIN {X -60.6837,Y -94.0883,Z 114,A -125.9687,B 24.9505,C -1.6252,E1 24.9151,E2 211.8096} C_DIS
LIN {X -57.6412,Y -95.9839,Z 114,A -124.1496,B 24.9507,C -1.6218,E1 24.9195,E2 209.993} C_DIS
LIN {X -54.4868,Y -97.8072,Z 114,A -122.4977,B 24.9514,C -1.6104,E1 24.9234,E2 208.3633} C_DIS
LIN {X -51.073,Y -99.6324,Z 114,A -120.5348,B 24.9516,C -1.6071,E1 24.9283,E2 206.4029} C_DIS
LIN {X -48.221,Y -101.044,Z 114,A -118.9164,B 24.9518,C -1.6047,E1 24.9323,E2 204.786} C_DIS
LIN {X -44.8368,Y -102.5901,Z 114,A -116.7372,B 24.9512,C -1.614,E1 24.9379,E2 202.5794} C_DIS
LIN {X -40.7257,Y -104.2906,Z 114,A -114.898,B 24.9524,C -1.5935,E1 24.9426,E2 200.7849} C_DIS
LIN {X -38.2437,Y -105.2259,Z 114,A -113.3235,B 24.952,C -1.6013,E1 24.9468,E2 199.1886} C_DIS
LIN {X -32.9889,Y -106.9898,Z 114,A -110.5337,B 24.9522,C -1.5971,E1 24.9542,E2 196.4037} C_DIS
LIN {X -29.919,Y -107.8902,Z 114,A -108.9232,B 24.9523,C -1.5948,E1 24.9585,E2 194.796} C_DIS
LIN {X -26.5998,Y -108.7544,Z 114,A -107.0678,B 24.9521,C -1.5981,E1 24.9635,E2 192.9302} C_DIS
LIN {X -22.9085,Y -109.5921,Z 114,A -105.1056,B 24.9521,C -1.5982,E1 24.9689,E2 190.9652} C_DIS
LIN {X -19.6259,Y -110.2267,Z 114,A -103.4597,B 24.9523,C -1.5948,E1 24.9734,E2 189.3256} C_DIS
LIN {X -15.3688,Y -110.9009,Z 114,A -101.2952,B 24.9525,C -1.5925,E1 24.9794,E2 187.1647} C_DIS
LIN {X -12.3542,Y -111.2774,Z 114,A -99.684,B 24.9524,C -1.5947,E1 24.9838,E2 185.5473} C_DIS
LIN {X -10.0088,Y -111.5122,Z 114,A -98.4207,B 24.9522,C -1.597,E1 24.9874,E2 184.2778} C_DIS
LIN {X -5.0158,Y -111.8479,Z 114,A -95.8508,B 24.9522,C -1.5975,E1 24.9945,E2 181.706} C_DIS
LIN {X 0.7944,Y -111.9312,Z 114,A -93.841,B 24.9546,C -1.5572,E1 25,E2 179.7915} C_DIS
Enddeposition()
LIN {X 0.7944,Y -111.9312,Z 114,A -93.841,B 24.9546,C -1.5572,E1 25,E2 179.7915} C_DIS
Startdeposition()
$VEL.CP = VEL_PRINT
LIN {X -2.4185,Y -111.0154,Z 114,A -95.2418,B 24.953,C -1.5835,E1 24.9962,E2 181.1301} C_DIS
LIN {X -6.4005,Y -110.8569,Z 114,A -97.5062,B 24.9535,C -1.5746,E1 24.9898,E2 183.4161} C_DIS
LIN {X -10.3207,Y -110.5605,Z 114,A -99.1908,B 24.9527,C -1.5891,E1 24.9852,E2 185.0672} C_DIS
LIN {X -13.392,Y -110.2317,Z 114,A -101.3383,B 24.954,C -1.5662,E1 24.9791,E2 187.2703} C_DIS
LIN {X -18.0578,Y -109.5633,Z 114,A -103.5259,B 24.9534,C -1.577,E1 24.9731,E2 189.4342} C_DIS
LIN {X -21.2893,Y -108.9816,Z 114,A -105.2444,B 24.9534,C -1.5766,E1 24.9684,E2 191.1555} C_DIS
LIN {X -24.6415,Y -108.2731,Z 114,A -107.0596,B 24.9534,C -1.5755,E1 24.9634,E2 192.9756} C_DIS
LIN {X -28.2112,Y -107.3993,Z 114,A -108.7885,B 24.953,C -1.5834,E1 24.9588,E2 194.6881} C_DIS
LIN {X -31.2122,Y -106.5649,Z 114,A -110.3239,B 24.9528,C -1.5874,E1 24.9547,E2 196.2164} C_DIS
LIN {X -36.9383,Y -104.7174,Z 114,A -113.3962,B 24.9526,C -1.5912,E1 24.9465,E2 199.2854} C_DIS
LIN {X -42.9682,Y -102.3909,Z 114,A -116.9361,B 24.9529,C -1.586,E1 24.9373,E2 202.8452} C_DIS
LIN {X -46.0927,Y -101.0241,Z 114,A -118.8197,B 24.9531,C -1.5829,E1 24.9324,E2 204.7407} C_DIS
LIN {X -49.1573,Y -99.5677,Z 114,A -120.533,B 24.9528,C -1.5866,E1 24.9281,E2 206.4497} C_DIS
LIN {X -52.5318,Y -97.8303,Z 114,A -122.5099,B 24.9528,C -1.5884,E1 24.9232,E2 208.4278} C_DIS
LIN {X -57.1043,Y -95.2348,Z 114,A -125.4107,B 24.9529,C -1.5848,E1 24.9162,E2 211.346} C_DIS
LIN {X -61.0625,Y -92.7444,Z 114,A -127.4244,B 24.9518,C -1.6045,E1 24.9116,E2 213.3191} C_DIS
LIN {X -65.8161,Y -89.434,Z 114,A -130.6019,B 24.9519,C -1.602,E1 24.9043,E2 216.5136} C_DIS
LIN {X -68.7684,Y -87.184,Z 114,A -132.7907,B 24.9524,C -1.5946,E1 24.8994,E2 218.7279} C_DIS
LIN {X -72.5215,Y -84.0905,Z 114,A -135.1394,B 24.9517,C -1.6058,E1 24.8944,E2 221.0592} C_DIS
LIN {X -75.5379,Y -81.3914,Z 114,A -137.1661,B 24.9513,C -1.6124,E1 24.8903,E2 223.0782} C_DIS
LIN {X -78.086,Y -78.9476,Z 114,A -138.9493,B 24.951,C -1.6178,E1 24.8867,E2 224.8561} C_DIS
LIN {X -80.6881,Y -76.2867,Z 114,A -140.8908,B 24.9508,C -1.6212,E1 24.8829,E2 226.7979} C_DIS
LIN {X -82.9924,Y -73.7737,Z 114,A -142.6466,B 24.9505,C -1.6253,E1 24.8796,E2 228.5518} C_DIS
LIN {X -85.5932,Y -70.7391,Z 114,A -144.7767,B 24.9504,C -1.6274,E1 24.8758,E2 230.6865} C_DIS
LIN {X -87.3619,Y -68.5433,Z 114,A -146.9968,B 24.952,C -1.6013,E1 24.8719,E2 232.9792} C_DIS
LIN {X -90.4148,Y -64.4616,Z 114,A -148.814,B 24.9496,C -1.6393,E1 24.869,E2 234.715} C_DIS
LIN {X -93.8367,Y -59.3736,Z 114,A -152.0396,B 24.9493,C -1.645,E1 24.8641,E2 237.943} C_DIS
LIN {X -95.6011,Y -56.4852,Z 114,A -153.7495,B 24.9489,C -1.6511,E1 24.8616,E2 239.6472} C_DIS
LIN {X -96.9832,Y -54.0777,Z 114,A -155.6163,B 24.9497,C -1.6383,E1 24.859,E2 241.5543} C_DIS
LIN {X -98.6138,Y -51.0447,Z 114,A -157.1898,B 24.9489,C -1.651,E1 24.857,E2 243.106} C_DIS
LIN {X -100.8299,Y -46.5146,Z 114,A -159.9191,B 24.9488,C -1.6535,E1 24.8537,E2 245.8441} C_DIS
LIN {X -102.7112,Y -42.198,Z 114,A -162.0537,B 24.9476,C -1.6718,E1 24.8514,E2 247.9468} C_DIS
LIN {X -103.8062,Y -39.4262,Z 114,A -163.6153,B 24.9474,C -1.6755,E1 24.8499,E2 249.5085} C_DIS
LIN {X -105.0185,Y -36.0785,Z 114,A -165.4899,B 24.9471,C -1.6795,E1 24.8481,E2 251.3842} C_DIS
LIN {X -106.2064,Y -32.4125,Z 114,A -168.1149,B 24.9483,C -1.6613,E1 24.8459,E2 254.0675} C_DIS
LIN {X -107.4239,Y -28.1155,Z 114,A -169.6399,B 24.946,C -1.698,E1 24.8449,E2 255.5139} C_DIS
LIN {X -108.6078,Y -23.1253,Z 114,A -172.5268,B 24.946,C -1.697,E1 24.843,E2 258.4201} C_DIS
LIN {X -109.3268,Y -19.4378,Z 114,A -174.8144,B 24.9465,C -1.6899,E1 24.8419,E2 260.7382} C_DIS
LIN {X -109.8846,Y -15.9894,Z 114,A -176.5416,B 24.9459,C -1.6985,E1 24.8412,E2 262.4553} C_DIS
LIN {X -110.4327,Y -11.6084,Z 114,A -178.4973,B 24.9447,C -1.718,E1 24.8406,E2 264.3762} C_DIS
LIN {X -110.7392,Y -8.207,Z 114,A 179.4619,B 24.945,C -1.7131,E1 24.8401,E2 266.441} C_DIS
LIN {X -111.0142,Y -2.4864,Z 114,A 176.668,B 24.944,C -1.7287,E1 24.8398,E2 269.2143} C_DIS
LIN {X -111.0337,Y 1.4247,Z 114,A 174.8211,B 24.9431,C -1.7418,E1 24.8398,E2 271.0413} C_DIS
LIN {X -110.9009,Y 5.6045,Z 114,A 172.6901,B 24.9426,C -1.7498,E1 24.84,E2 273.166} C_DIS
LIN {X -110.5821,Y 10.087,Z 114,A 170.2436,B 24.9424,C -1.7525,E1 24.8406,E2 275.6208} C_DIS
LIN {X -110.2205,Y 13.4877,Z 114,A 168.4615,B 24.9421,C -1.7575,E1 24.8411,E2 277.4015} C_DIS
LIN {X -109.8192,Y 16.4367,Z 114,A 166.6911,B 24.9424,C -1.7536,E1 24.8418,E2 279.1918} C_DIS
LIN {X -108.4112,Y 24.0268,Z 114,A 161.8404,B 24.9436,C -1.734,E1 24.8446,E2 284.1179} C_DIS
LIN {X -106.9445,Y 29.8859,Z 114,A 159.9418,B 24.94,C -1.7897,E1 24.8459,E2 285.8948} C_DIS
LIN {X -105.4534,Y 34.7868,Z 114,A 157.0163,B 24.9401,C -1.7872,E1 24.8483,E2 288.8429} C_DIS
LIN {X -104.3889,Y 37.8569,Z 114,A 155.0611,B 24.9405,C -1.782,E1 24.8502,E2 290.8217} C_DIS
LIN {X -102.914,Y 41.6998,Z 114,A 152.5354,B 24.9411,C -1.7734,E1 24.8529,E2 293.382} C_DIS
LIN {X -101.0499,Y 46.0354,Z 114,A 150.738,B 24.9389,C -1.8048,E1 24.8548,E2 295.1143} C_DIS
LIN {X -99.4223,Y 49.4507,Z 114,A 148.8226,B 24.9385,C -1.8121,E1 24.8572,E2 297.0228} C_DIS
LIN {X -97.6613,Y 52.8433,Z 114,A 146.8025,B 24.9382,C -1.8161,E1 24.8598,E2 299.0441} C_DIS
LIN {X -95.5143,Y 56.632,Z 114,A 144.0848,B 24.9389,C -1.8048,E1 24.8637,E2 301.8028} C_DIS
LIN {X -93.5278,Y 59.8557,Z 114,A 142.1394,B 24.9385,C -1.8106,E1 24.8666,E2 303.7442} C_DIS
LIN {X -91.4508,Y 62.9851,Z 114,A 140.6905,B 24.9369,C -1.8347,E1 24.8688,E2 305.143} C_DIS
LIN {X -88.605,Y 66.9281,Z 114,A 137.9517,B 24.937,C -1.8327,E1 24.8734,E2 307.8996} C_DIS
LIN {X -83.8614,Y 72.7841,Z 114,A 134.2305,B 24.9359,C -1.8493,E1 24.8799,E2 311.5984} C_DIS
LIN {X -82.0228,Y 74.8498,Z 114,A 132.1325,B 24.9374,C -1.8273,E1 24.884,E2 313.7583} C_DIS
LIN {X -78.9433,Y 78.0903,Z 114,A 129.868,B 24.9369,C -1.8345,E1 24.8884,E2 316.0152} C_DIS
LIN {X -75.8797,Y 81.0709,Z 114,A 128.1943,B 24.9351,C -1.8602,E1 24.8917,E2 317.6347} C_DIS
LIN {X -73.2325,Y 83.4698,Z 114,A 125.918,B 24.936,C -1.8477,E1 24.8966,E2 319.9497} C_DIS
LIN {X -70.3255,Y 85.9345,Z 114,A 123.5631,B 24.9367,C -1.8372,E1 24.9017,E2 322.3386} C_DIS
LIN {X -66.0869,Y 89.2358,Z 114,A 121.7581,B 24.9337,C -1.8803,E1 24.9055,E2 324.0474} C_DIS
LIN {X -61.9172,Y 92.1768,Z 114,A 118.653,B 24.9346,C -1.8672,E1 24.9128,E2 327.1941} C_DIS
LIN {X -57.8305,Y 94.7935,Z 114,A 116.5411,B 24.9332,C -1.8872,E1 24.9177,E2 329.2651} C_DIS
LIN {X -55.0825,Y 96.4164,Z 114,A 114.9095,B 24.933,C -1.8908,E1 24.9216,E2 330.8931} C_DIS
LIN {X -49.1383,Y 99.5771,Z 114,A 111.2974,B 24.933,C -1.8912,E1 24.9306,E2 334.5143} C_DIS
LIN {X -45.7232,Y 101.1906,Z 114,A 109.4315,B 24.9325,C -1.8974,E1 24.9352,E2 336.3699} C_DIS
LIN {X -39.3598,Y 103.8313,Z 114,A 105.9254,B 24.932,C -1.9043,E1 24.9443,E2 339.8674} C_DIS
LIN {X -36.5002,Y 104.8711,Z 114,A 103.4862,B 24.9343,C -1.8719,E1 24.951,E2 342.3884} C_DIS
LIN {X -31.8162,Y 106.3857,Z 114,A 101.9855,B 24.9312,C -1.9161,E1 24.9547,E2 343.7867} C_DIS
LIN {X -26.8818,Y 107.7397,Z 114,A 98.9867,B 24.932,C -1.9044,E1 24.9629,E2 346.8179} C_DIS
LIN {X -23.3175,Y 108.5659,Z 114,A 97.1017,B 24.9319,C -1.9062,E1 24.968,E2 348.701} C_DIS
LIN {X -18.8805,Y 109.4258,Z 114,A 94.8136,B 24.9316,C -1.9098,E1 24.9742,E2 350.983} C_DIS
LIN {X -15.665,Y 109.9306,Z 114,A 93.1658,B 24.9314,C -1.9122,E1 24.9788,E2 352.6264} C_DIS
LIN {X -12.1993,Y 110.3709,Z 114,A 91.2301,B 24.9318,C -1.9078,E1 24.9842,E2 354.5738} C_DIS
LIN {X -8.5865,Y 110.709,Z 114,A 89.385,B 24.9316,C -1.9098,E1 24.9893,E2 356.4151} C_DIS
LIN {X -4.8889,Y 110.9335,Z 114,A 87.797,B 24.9306,C -1.9238,E1 24.9936,E2 357.9705} C_DIS
LIN {X -0.4832,Y 111.0403,Z 114,A 85.28,B 24.9313,C -1.9144,E1 25.0007,E2 360.5099} C_DIS
LIN {X 3.5071,Y 110.9858,Z 114,A 83.1984,B 24.9313,C -1.9137,E1 25.0065,E2 362.5928} C_DIS
LIN {X 7.1517,Y 110.8111,Z 114,A 81.3183,B 24.9313,C -1.9138,E1 25.0118,E2 364.4718} C_DIS
LIN {X 10.5655,Y 110.5379,Z 114,A 79.4848,B 24.9315,C -1.9109,E1 25.0169,E2 366.3111} C_DIS
LIN {X 14.1795,Y 110.1321,Z 114,A 77.6988,B 24.9313,C -1.9143,E1 25.0218,E2 368.0877} C_DIS
LIN {X 17.817,Y 109.6036,Z 114,A 75.7174,B 24.9316,C -1.9102,E1 25.0273,E2 370.077} C_DIS
LIN {X 21.1526,Y 109.0079,Z 114,A 74.1008,B 24.9312,C -1.915,E1 25.0317,E2 371.6804} C_DIS
LIN {X 24.6005,Y 108.2826,Z 114,A 72.3306,B 24.9312,C -1.9161,E1 25.0365,E2 373.4457} C_DIS
LIN {X 28.3244,Y 107.3699,Z 114,A 70.3483,B 24.9312,C -1.9147,E1 25.0419,E2 375.4283} C_DIS
LIN {X 33.9328,Y 105.7297,Z 114,A 67.5221,B 24.9309,C -1.9205,E1 25.0495,E2 378.2361} C_DIS
LIN {X 39.9901,Y 103.5923,Z 114,A 63.8412,B 24.9322,C -1.9019,E1 25.0592,E2 381.9534} C_DIS
LIN {X 43.3049,Y 102.249,Z 114,A 62.0608,B 24.9322,C -1.9027,E1 25.0638,E2 383.7277} C_DIS
LIN {X 46.8633,Y 100.6676,Z 114,A 60.1123,B 24.9322,C -1.903,E1 25.0687,E2 385.6707} C_DIS
LIN {X 49.9423,Y 99.1783,Z 114,A 58.2287,B 24.9326,C -1.8957,E1 25.0735,E2 387.5665} C_DIS
LIN {X 54.7707,Y 96.5956,Z 114,A 55.2186,B 24.9335,C -1.8839,E1 25.0809,E2 390.5958} C_DIS
LIN {X 58.6973,Y 94.2592,Z 114,A 52.5403,B 24.9347,C -1.8667,E1 25.0873,E2 393.3063} C_DIS
LIN {X 62.3596,Y 91.8773,Z 114,A 50.9273,B 24.933,C -1.8904,E1 25.0909,E2 394.858} C_DIS
LIN {X 65.3934,Y 89.7435,Z 114,A 49.0471,B 24.9331,C -1.8885,E1 25.0952,E2 396.7359} C_DIS
LIN {X 67.8047,Y 87.9356,Z 114,A 47.4821,B 24.9334,C -1.8853,E1 25.0987,E2 398.3029} C_DIS
LIN {X 71.5005,Y 84.9604,Z 114,A 44.9272,B 24.934,C -1.876,E1 25.1042,E2 400.8701} C_DIS
LIN {X 74.1243,Y 82.6785,Z 114,A 43.3962,B 24.9335,C -1.8839,E1 25.1074,E2 402.3763} C_DIS
LIN {X 76.7486,Y 80.2494,Z 114,A 41.377,B 24.9343,C -1.8724,E1 25.1115,E2 404.4142} C_DIS
LIN {X 79.3428,Y 77.6859,Z 114,A 38.7861,B 24.9367,C -1.8376,E1 25.1167,E2 407.0762} C_DIS
LIN {X 82.6441,Y 74.1627,Z 114,A 37.0944,B 24.9347,C -1.8667,E1 25.1198,E2 408.6918} C_DIS
LIN {X 84.6555,Y 71.8584,Z 114,A 35.5032,B 24.935,C -1.8625,E1 25.1227,E2 410.2858} C_DIS
LIN {X 87.5405,Y 68.316,Z 114,A 32.8954,B 24.9361,C -1.8458,E1 25.1273,E2 412.9208} C_DIS
LIN {X 90.1027,Y 64.8991,Z 114,A 30.8983,B 24.9359,C -1.8494,E1 25.1305,E2 414.8999} C_DIS
LIN {X 91.9846,Y 62.2011,Z 114,A 29.2815,B 24.9359,C -1.8486,E1 25.1331,E2 416.5106} C_DIS
LIN {X 94.0093,Y 59.0973,Z 114,A 26.8523,B 24.9379,C -1.8208,E1 25.1368,E2 418.9931} C_DIS
LIN {X 96.0192,Y 55.7738,Z 114,A 25.514,B 24.9362,C -1.8448,E1 25.1386,E2 420.268} C_DIS
LIN {X 97.9968,Y 52.2213,Z 114,A 23.202,B 24.9373,C -1.8295,E1 25.1417,E2 422.6039} C_DIS
LIN {X 99.611,Y 49.07,Z 114,A 21.4494,B 24.9373,C -1.8277,E1 25.1439,E2 424.3515} C_DIS
LIN {X 101.104,Y 45.9154,Z 114,A 19.6611,B 24.9377,C -1.8231,E1 25.146,E2 426.1409} C_DIS
LIN {X 102.4426,Y 42.8455,Z 114,A 17.4453,B 24.9395,C -1.7964,E1 25.1485,E2 428.4074} C_DIS
LIN {X 103.8634,Y 39.2751,Z 114,A 15.414,B 24.9401,C -1.7884,E1 25.1505,E2 430.4463} C_DIS
LIN {X 105.2516,Y 35.387,Z 114,A 12.8813,B 24.9417,C -1.7643,E1 25.1528,E2 433.0216} C_DIS
LIN {X 107.0029,Y 29.68,Z 114,A 10.7592,B 24.9395,C -1.7972,E1 25.1543,E2 435.0539} C_DIS
LIN {X 107.8691,Y 26.3515,Z 114,A 9.096,B 24.9395,C -1.7968,E1 25.1555,E2 436.7086} C_DIS
LIN {X 108.5792,Y 23.2567,Z 114,A 7.348,B 24.9402,C -1.7867,E1 25.1565,E2 438.4701} C_DIS
LIN {X 109.291,Y 19.6369,Z 114,A 5.548,B 24.9402,C -1.7854,E1 25.1575,E2 440.2627} C_DIS
LIN {X 109.8882,Y 15.9635,Z 114,A 3.6,B 24.9407,C -1.778,E1 25.1583,E2 442.2166} C_DIS
LIN {X 110.3432,Y 12.44,Z 114,A 1.6966,B 24.9413,C -1.769,E1 25.1589,E2 444.1301} C_DIS
LIN {X 110.6985,Y 8.7178,Z 114,A -0.1029,B 24.9413,C -1.7686,E1 25.1594,E2 445.9198} C_DIS
LIN {X 110.9359,Y 4.8348,Z 114,A -1.93,B 24.9413,C -1.7703,E1 25.1597,E2 447.7322} C_DIS
LIN {X 111.0231,Y 2.004,Z 114,A -3.9872,B 24.9433,C -1.7388,E1 25.1597,E2 449.8514} C_DIS
LIN {X 111.0312,Y -1.5643,Z 114,A -5.4186,B 24.9425,C -1.7511,E1 25.1597,E2 451.2452} C_DIS
LIN {X 110.9436,Y -4.6545,Z 114,A -6.9081,B 24.9425,C -1.7507,E1 25.1597,E2 452.7268} C_DIS
LIN {X 110.4115,Y -11.8112,Z 114,A -10.672,B 24.9435,C -1.7359,E1 25.1588,E2 456.5033} C_DIS
LIN {X 109.9628,Y -15.4386,Z 114,A -12.5228,B 24.9438,C -1.7313,E1 25.1581,E2 458.3539} C_DIS
LIN {X 109.3991,Y -19.0357,Z 114,A -14.3753,B 24.9441,C -1.7264,E1 25.1572,E2 460.2072} C_DIS
LIN {X 108.8101,Y -22.1481,Z 114,A -16.054,B 24.9446,C -1.7191,E1 25.1563,E2 461.8931} C_DIS
LIN {X 107.9859,Y -25.8725,Z 114,A -18.3061,B 24.9458,C -1.7001,E1 25.1549,E2 464.1772} C_DIS
LIN {X 106.9539,Y -29.853,Z 114,A -20.842,B 24.9474,C -1.6748,E1 25.153,E2 466.7581} C_DIS
LIN {X 105.5121,Y -34.6053,Z 114,A -22.7241,B 24.946,C -1.6971,E1 25.1514,E2 468.577} C_DIS
LIN {X 104.0831,Y -38.695,Z 114,A -25.5183,B 24.948,C -1.6651,E1 25.1487,E2 471.431} C_DIS
LIN {X 102.4296,Y -42.8763,Z 114,A -27.1486,B 24.9466,C -1.6887,E1 25.147,E2 472.9965} C_DIS
LIN {X 101.1616,Y -45.7876,Z 114,A -28.7621,B 24.9468,C -1.6849,E1 25.1452,E2 474.6104} C_DIS
LIN {X 98.8745,Y -50.5367,Z 114,A -32.1776,B 24.9493,C -1.6456,E1 25.1408,E2 478.1001} C_DIS
LIN {X 96.6091,Y -54.7472,Z 114,A -33.8463,B 24.9475,C -1.6739,E1 25.1387,E2 479.6935} C_DIS
LIN {X 94.4598,Y -58.3747,Z 114,A -36.3664,B 24.9488,C -1.6522,E1 25.135,E2 482.2518} C_DIS
LIN {X 90.7957,Y -63.9275,Z 114,A -39.6195,B 24.949,C -1.6505,E1 25.1299,E2 485.4929} C_DIS
LIN {X 88.5593,Y -66.989,Z 114,A -41.5564,B 24.9492,C -1.6461,E1 25.1267,E2 487.4311} C_DIS
LIN {X 86.2551,Y -69.9299,Z 114,A -43.345,B 24.9492,C -1.6471,E1 25.1236,E2 489.2088} C_DIS
LIN {X 83.9302,Y -72.7053,Z 114,A -45.2374,B 24.9495,C -1.6411,E1 25.1201,E2 491.1067} C_DIS
LIN {X 81.7749,Y -75.12,Z 114,A -46.8671,B 24.9497,C -1.6386,E1 25.1171,E2 492.7351} C_DIS
LIN {X 79.1971,Y -77.8334,Z 114,A -48.8066,B 24.95,C -1.6334,E1 25.1133,E2 494.6785} C_DIS
LIN {X 76.8504,Y -80.1514,Z 114,A -50.4619,B 24.9501,C -1.6314,E1 25.11,E2 496.3318} C_DIS
LIN {X 74.3249,Y -82.4989,Z 114,A -52.2536,B 24.9504,C -1.6266,E1 25.1063,E2 498.1274} C_DIS
LIN {X 71.9166,Y -84.6059,Z 114,A -53.9281,B 24.9507,C -1.6218,E1 25.1028,E2 499.8068} C_DIS
LIN {X 68.9916,Y -87.0077,Z 114,A -56.0802,B 24.9515,C -1.6087,E1 25.098,E2 501.9816} C_DIS
LIN {X 65.2846,Y -89.8232,Z 114,A -58.3426,B 24.9515,C -1.6097,E1 25.093,E2 504.2335} C_DIS
LIN {X 62.0134,Y -92.1117,Z 114,A -60.0636,B 24.9508,C -1.6204,E1 25.0891,E2 505.9233} C_DIS
LIN {X 59.2228,Y -93.9309,Z 114,A -62.7892,B 24.9536,C -1.5732,E1 25.0824,E2 508.7518} C_DIS
LIN {X 54.9136,Y -96.5135,Z 114,A -64.4776,B 24.9516,C -1.6077,E1 25.0786,E2 510.3536} C_DIS
LIN {X 48.1227,Y -100.0717,Z 114,A -68.5569,B 24.9523,C -1.5956,E1 25.0684,E2 514.4502} C_DIS
LIN {X 44.7284,Y -101.6349,Z 114,A -71.197,B 24.9543,C -1.5619,E1 25.0615,E2 517.1635} C_DIS
LIN {X 40.2422,Y -103.4932,Z 114,A -73.031,B 24.9528,C -1.5872,E1 25.0569,E2 518.9335} C_DIS
LIN {X 36.8046,Y -104.7643,Z 114,A -74.8484,B 24.9528,C -1.5879,E1 25.0521,E2 520.7456} C_DIS
LIN {X 33.116,Y -105.9883,Z 114,A -76.5574,B 24.9521,C -1.5982,E1 25.0477,E2 522.4269} C_DIS
LIN {X 28.0673,Y -107.4363,Z 114,A -79.599,B 24.9532,C -1.5809,E1 25.0394,E2 525.5044} C_DIS
LIN {X 24.6784,Y -108.2646,Z 114,A -81.2981,B 24.953,C -1.5835,E1 25.0348,E2 527.195} C_DIS
LIN {X 21.2278,Y -108.9935,Z 114,A -83.2224,B 24.9534,C -1.5774,E1 25.0295,E2 529.1312} C_DIS
LIN {X 17.3457,Y -109.6787,Z 114,A -85.2344,B 24.9534,C -1.5768,E1 25.024,E2 531.1426} C_DIS
LIN {X 13.9102,Y -110.167,Z 114,A -86.8798,B 24.9531,C -1.5818,E1 25.0194,E2 532.7748} C_DIS
LIN {X 8.5139,Y -110.7148,Z 114,A -90.0871,B 24.9542,C -1.563,E1 25.0104,E2 536.0246} C_DIS
LIN {X 3.6446,Y -110.9816,Z 114,A -92.2781,B 24.9535,C -1.5758,E1 25.0044,E2 538.1848} C_DIS
LIN {X 0.7959,Y -111.0208,Z 114,A -93.8182,B 24.9537,C -1.5727,E1 25.0001,E2 539.732} C_DIS
Enddeposition()
LIN {X 0.7959,Y -111.0208,Z 114,A -93.8182,B 24.9537,C -1.5727,E1 25.0001,E2 539.732} C_DIS
Startdeposition()
$VEL.CP = VEL_PRINT
LIN {X 1.5789,Y -110.1118,Z 114,A -92.6168,B 24.9507,C -1.622,E1 25.0037,E2 538.4139} C_DIS
LIN {X 4.9385,Y -110.0116,Z 114,A -90.8561,B 24.9507,C -1.6232,E1 25.0087,E2 536.6509} C_DIS
LIN {X 7.7428,Y -109.8501,Z 114,A -89.3371,B 24.9504,C -1.6263,E1 25.0129,E2 535.1253} C_DIS
LIN {X 12.8337,Y -109.3719,Z 114,A -86.7608,B 24.9506,C -1.6242,E1 25.0201,E2 532.5555} C_DIS
LIN {X 16.324,Y -108.9068,Z 114,A -84.8476,B 24.9503,C -1.6289,E1 25.0254,E2 530.6329} C_DIS
LIN {X 19.443,Y -108.3922,Z 114,A -83.252,B 24.9503,C -1.6281,E1 25.0297,E2 529.0409} C_DIS
LIN {X 22.9274,Y -107.7105,Z 114,A -81.3643,B 24.9501,C -1.6314,E1 25.0349,E2 527.1477} C_DIS
LIN {X 26.098,Y -106.985,Z 114,A -79.7227,B 24.9501,C -1.6309,E1 25.0394,E2 525.5096} C_DIS
Enddeposition()
END
